	VAR robtarget Openhole_4834 := [[446.33, -4.29, 181.85], [-0.058838, 0.704655, 0.706057, -0.038517], [0,0,0,0], [9E9, 9E9, 9E9, 9E9, 9E9, 9E9]];
	VAR robtarget Openhole_4835 := [[445.84, -4.38, 181.92], [-0.060204, 0.704539, 0.70616, -0.036572], [0,0,0,0], [9E9, 9E9, 9E9, 9E9, 9E9, 9E9]];
	VAR robtarget Openhole_4836 := [[444.87, -4.57, 182.04], [-0.062827, 0.70431, 0.706355, -0.032605], [0,0,0,0], [9E9, 9E9, 9E9, 9E9, 9E9, 9E9]];
	VAR robtarget Openhole_4837 := [[438.56, -5.94, 182.78], [-0.079375, 0.702638, 0.707077, -0.006541], [0,0,0,0], [9E9, 9E9, 9E9, 9E9, 9E9, 9E9]];
	VAR robtarget Openhole_4838 := [[432.17, -6.93, 183.42], [-0.097021, 0.700419, 0.706868, 0.018385], [0,0,0,0], [9E9, 9E9, 9E9, 9E9, 9E9, 9E9]];
	VAR robtarget Openhole_4839 := [[431.68, -6.99, 183.47], [-0.09841, 0.700225, 0.706817, 0.020252], [0,0,0,0], [9E9, 9E9, 9E9, 9E9, 9E9, 9E9]];
	VAR robtarget Openhole_4840 := [[437.22, -4.54, 183.11], [-0.088439, 0.701554, 0.707076, -0.00665], [0,0,0,0], [9E9, 9E9, 9E9, 9E9, 9E9, 9E9]];
	VAR robtarget Openhole_4841 := [[442.51, -3.16, 182.47], [-0.075483, 0.703066, 0.706502, -0.029244], [0,0,0,0], [9E9, 9E9, 9E9, 9E9, 9E9, 9E9]];
	VAR robtarget Openhole_4842 := [[444.89, -2.47, 182.13], [-0.069759, 0.703657, 0.705995, -0.039633], [0,0,0,0], [9E9, 9E9, 9E9, 9E9, 9E9, 9E9]];
	VAR robtarget Openhole_4843 := [[445.84, -2.22, 181.99], [-0.067345, 0.703893, 0.705754, -0.043713], [0,0,0,0], [9E9, 9E9, 9E9, 9E9, 9E9, 9E9]];
	VAR robtarget Openhole_4844 := [[446.81, -2.01, 181.84], [-0.064778, 0.704133, 0.705496, -0.047696], [0,0,0,0], [9E9, 9E9, 9E9, 9E9, 9E9, 9E9]];
	VAR robtarget Openhole_4845 := [[447.3, -1.93, 181.76], [-0.063421, 0.704257, 0.705363, -0.049635], [0,0,0,0], [9E9, 9E9, 9E9, 9E9, 9E9, 9E9]];
	VAR robtarget Openhole_4846 := [[447.78, -1.85, 181.68], [-0.06202, 0.704382, 0.705226, -0.051544], [0,0,0,0], [9E9, 9E9, 9E9, 9E9, 9E9, 9E9]];
	VAR robtarget Openhole_4847 := [[448.27, -1.79, 181.6], [-0.060567, 0.704508, 0.705087, -0.053411], [0,0,0,0], [9E9, 9E9, 9E9, 9E9, 9E9, 9E9]];
	VAR robtarget Openhole_4848 := [[448.77, -1.75, 181.52], [-0.059016, 0.70464, 0.704949, -0.055201], [0,0,0,0], [9E9, 9E9, 9E9, 9E9, 9E9, 9E9]];
	VAR robtarget Openhole_4849 := [[449.26, -1.74, 181.44], [-0.057379, 0.704775, 0.704813, -0.056912], [0,0,0,0], [9E9, 9E9, 9E9, 9E9, 9E9, 9E9]];
	VAR robtarget Openhole_4850 := [[449.75, -1.74, 181.35], [-0.055693, 0.70491, 0.704677, -0.058572], [0,0,0,0], [9E9, 9E9, 9E9, 9E9, 9E9, 9E9]];
	VAR robtarget Openhole_4851 := [[450.24, -1.78, 181.27], [-0.053891, 0.70505, 0.704547, -0.060109], [0,0,0,0], [9E9, 9E9, 9E9, 9E9, 9E9, 9E9]];
	VAR robtarget Openhole_4852 := [[450.74, -1.83, 181.19], [-0.05205, 0.705189, 0.704419, -0.061598], [0,0,0,0], [9E9, 9E9, 9E9, 9E9, 9E9, 9E9]];
	VAR robtarget Openhole_4853 := [[451.22, -1.9, 181.11], [-0.050156, 0.705326, 0.704293, -0.063023], [0,0,0,0], [9E9, 9E9, 9E9, 9E9, 9E9, 9E9]];
	VAR robtarget Openhole_4854 := [[456.58, -2.86, 180.3], [-0.028679, 0.706525, 0.702811, -0.077823], [0,0,0,0], [9E9, 9E9, 9E9, 9E9, 9E9, 9E9]];
	VAR robtarget Openhole_4855 := [[458.54, -3.07, 180.01], [-0.021229, 0.706788, 0.702142, -0.083644], [0,0,0,0], [9E9, 9E9, 9E9, 9E9, 9E9, 9E9]];
	VAR robtarget Openhole_4856 := [[459.53, -3.13, 179.86], [-0.01766, 0.706886, 0.701769, -0.086718], [0,0,0,0], [9E9, 9E9, 9E9, 9E9, 9E9, 9E9]];
	VAR robtarget Openhole_4857 := [[460.52, -3.16, 179.71], [-0.014191, 0.706964, 0.701371, -0.089885], [0,0,0,0], [9E9, 9E9, 9E9, 9E9, 9E9, 9E9]];
	VAR robtarget Openhole_4858 := [[461.02, -3.16, 179.64], [-0.012499, 0.706996, 0.701161, -0.091504], [0,0,0,0], [9E9, 9E9, 9E9, 9E9, 9E9, 9E9]];
	VAR robtarget Openhole_4859 := [[461.51, -3.15, 179.56], [-0.010815, 0.707024, 0.700947, -0.093127], [0,0,0,0], [9E9, 9E9, 9E9, 9E9, 9E9, 9E9]];
	VAR robtarget Openhole_4860 := [[466.44, -2.87, 178.76], [0.005029, 0.707089, 0.6985, -0.109988], [0,0,0,0], [9E9, 9E9, 9E9, 9E9, 9E9, 9E9]];
	VAR robtarget Openhole_4861 := [[473.81, -2.37, 177.5], [0.028255, 0.706542, 0.69417, -0.13464], [0,0,0,0], [9E9, 9E9, 9E9, 9E9, 9E9, 9E9]];
	VAR robtarget Openhole_4862 := [[476.77, -2.31, 177.01], [0.037899, 0.70609, 0.692338, -0.143766], [0,0,0,0], [9E9, 9E9, 9E9, 9E9, 9E9, 9E9]];
	VAR robtarget Openhole_4863 := [[477.26, -2.32, 176.93], [0.039535, 0.706001, 0.692031, -0.145236], [0,0,0,0], [9E9, 9E9, 9E9, 9E9, 9E9, 9E9]];
	VAR robtarget Openhole_4864 := [[482.7, -2.51, 176.12], [0.05787, 0.704735, 0.688645, -0.160526], [0,0,0,0], [9E9, 9E9, 9E9, 9E9, 9E9, 9E9]];
	VAR robtarget Openhole_4865 := [[489.12, -3.09, 175.32], [0.079987, 0.702568, 0.684666, -0.176726], [0,0,0,0], [9E9, 9E9, 9E9, 9E9, 9E9, 9E9]];
	VAR robtarget Openhole_4866 := [[495.54, -3.95, 174.71], [0.102089, 0.699698, 0.680767, -0.191199], [0,0,0,0], [9E9, 9E9, 9E9, 9E9, 9E9, 9E9]];
	VAR robtarget Openhole_4867 := [[495.59, -2.66, 174.13], [0.098369, 0.700231, 0.679658, -0.195101], [0,0,0,0], [9E9, 9E9, 9E9, 9E9, 9E9, 9E9]];
	VAR robtarget Openhole_4868 := [[489.19, -1.71, 174.77], [0.075928, 0.703018, 0.683527, -0.181082], [0,0,0,0], [9E9, 9E9, 9E9, 9E9, 9E9, 9E9]];
	VAR robtarget Openhole_4869 := [[483.28, -1.11, 175.57], [0.055318, 0.70494, 0.68723, -0.166476], [0,0,0,0], [9E9, 9E9, 9E9, 9E9, 9E9, 9E9]];
	VAR robtarget Openhole_4870 := [[477.85, -0.87, 176.44], [0.036842, 0.706146, 0.690683, -0.151515], [0,0,0,0], [9E9, 9E9, 9E9, 9E9, 9E9, 9E9]];
	VAR robtarget Openhole_4871 := [[476.87, -0.86, 176.61], [0.033562, 0.70631, 0.691313, -0.148613], [0,0,0,0], [9E9, 9E9, 9E9, 9E9, 9E9, 9E9]];
	VAR robtarget Openhole_4872 := [[476.37, -0.86, 176.69], [0.031934, 0.706385, 0.691629, -0.147139], [0,0,0,0], [9E9, 9E9, 9E9, 9E9, 9E9, 9E9]];
	VAR robtarget Openhole_4873 := [[470.48, -1.08, 177.77], [0.012862, 0.70699, 0.695336, -0.128482], [0,0,0,0], [9E9, 9E9, 9E9, 9E9, 9E9, 9E9]];
	VAR robtarget Openhole_4874 := [[462.62, -1.59, 179.19], [-0.012185, 0.707002, 0.699732, -0.10186], [0,0,0,0], [9E9, 9E9, 9E9, 9E9, 9E9, 9E9]];
	VAR robtarget Openhole_4875 := [[461.64, -1.61, 179.36], [-0.015476, 0.706937, 0.700202, -0.098575], [0,0,0,0], [9E9, 9E9, 9E9, 9E9, 9E9, 9E9]];
	VAR robtarget Openhole_4876 := [[461.14, -1.61, 179.44], [-0.017156, 0.706899, 0.700428, -0.096959], [0,0,0,0], [9E9, 9E9, 9E9, 9E9, 9E9, 9E9]];
	VAR robtarget Openhole_4877 := [[460.65, -1.61, 179.53], [-0.018855, 0.706855, 0.700648, -0.095356], [0,0,0,0], [9E9, 9E9, 9E9, 9E9, 9E9, 9E9]];
	VAR robtarget Openhole_4878 := [[460.16, -1.6, 179.61], [-0.020577, 0.706807, 0.700861, -0.093773], [0,0,0,0], [9E9, 9E9, 9E9, 9E9, 9E9, 9E9]];
	VAR robtarget Openhole_4879 := [[459.17, -1.56, 179.77], [-0.024104, 0.706696, 0.701268, -0.09068], [0,0,0,0], [9E9, 9E9, 9E9, 9E9, 9E9, 9E9]];
	VAR robtarget Openhole_4880 := [[457.2, -1.38, 180.09], [-0.031441, 0.706407, 0.702007, -0.084775], [0,0,0,0], [9E9, 9E9, 9E9, 9E9, 9E9, 9E9]];
	VAR robtarget Openhole_4881 := [[454.77, -0.99, 180.48], [-0.04106, 0.705914, 0.702801, -0.077911], [0,0,0,0], [9E9, 9E9, 9E9, 9E9, 9E9, 9E9]];
	VAR robtarget Openhole_4882 := [[453.8, -0.8, 180.64], [-0.045008, 0.705673, 0.703086, -0.075301], [0,0,0,0], [9E9, 9E9, 9E9, 9E9, 9E9, 9E9]];
	VAR robtarget Openhole_4883 := [[452.84, -0.58, 180.8], [-0.049026, 0.705405, 0.703349, -0.0728], [0,0,0,0], [9E9, 9E9, 9E9, 9E9, 9E9, 9E9]];
	VAR robtarget Openhole_4884 := [[451.9, -0.27, 180.96], [-0.053242, 0.705099, 0.703568, -0.070651], [0,0,0,0], [9E9, 9E9, 9E9, 9E9, 9E9, 9E9]];
	VAR robtarget Openhole_4885 := [[451.43, -0.1, 181.04], [-0.055377, 0.704935, 0.703669, -0.069639], [0,0,0,0], [9E9, 9E9, 9E9, 9E9, 9E9, 9E9]];
	VAR robtarget Openhole_4886 := [[450.48, 0.12, 181.21], [-0.059395, 0.704608, 0.703911, -0.067156], [0,0,0,0], [9E9, 9E9, 9E9, 9E9, 9E9, 9E9]];
	VAR robtarget Openhole_4887 := [[449.49, 0.16, 181.39], [-0.062852, 0.704308, 0.704209, -0.063946], [0,0,0,0], [9E9, 9E9, 9E9, 9E9, 9E9, 9E9]];
	VAR robtarget Openhole_4888 := [[448.52, 0, 181.57], [-0.065623, 0.704055, 0.704545, -0.060131], [0,0,0,0], [9E9, 9E9, 9E9, 9E9, 9E9, 9E9]];
	VAR robtarget Openhole_4889 := [[448.05, -0.13, 181.66], [-0.066822, 0.703942, 0.704716, -0.058103], [0,0,0,0], [9E9, 9E9, 9E9, 9E9, 9E9, 9E9]];
	VAR robtarget Openhole_4890 := [[447.57, -0.24, 181.74], [-0.068056, 0.703824, 0.704878, -0.056092], [0,0,0,0], [9E9, 9E9, 9E9, 9E9, 9E9, 9E9]];
	VAR robtarget Openhole_4891 := [[447.09, -0.38, 181.83], [-0.069208, 0.703712, 0.705039, -0.054033], [0,0,0,0], [9E9, 9E9, 9E9, 9E9, 9E9, 9E9]];
	VAR robtarget Openhole_4892 := [[446.14, -0.63, 181.99], [-0.071596, 0.703473, 0.70534, -0.049958], [0,0,0,0], [9E9, 9E9, 9E9, 9E9, 9E9, 9E9]];
	VAR robtarget Openhole_4893 := [[445.19, -0.91, 182.15], [-0.073903, 0.703234, 0.70562, -0.045831], [0,0,0,0], [9E9, 9E9, 9E9, 9E9, 9E9, 9E9]];
	VAR robtarget Openhole_4894 := [[439.03, -2.77, 183.04], [-0.088301, 0.701572, 0.706861, -0.01864], [0,0,0,0], [9E9, 9E9, 9E9, 9E9, 9E9, 9E9]];
	VAR robtarget Openhole_4895 := [[441.88, -4.7, 182.45], [-0.072446, 0.703386, 0.706765, -0.021976], [0,0,0,0], [9E9, 9E9, 9E9, 9E9, 9E9, 9E9]];
	VAR robtarget Openhole_4896 := [[444.74, -6.64, 181.97], [-0.056353, 0.704858, 0.706655, -0.025274], [0,0,0,0], [9E9, 9E9, 9E9, 9E9, 9E9, 9E9]];
	VAR robtarget Openhole_4897 := [[445.24, -6.56, 181.91], [-0.054946, 0.704969, 0.706583, -0.027199], [0,0,0,0], [9E9, 9E9, 9E9, 9E9, 9E9, 9E9]];
	VAR robtarget Openhole_4898 := [[446.22, -6.44, 181.8], [-0.052032, 0.70519, 0.706428, -0.030973], [0,0,0,0], [9E9, 9E9, 9E9, 9E9, 9E9, 9E9]];
	VAR robtarget Openhole_4899 := [[447.21, -6.37, 181.68], [-0.048911, 0.705413, 0.706261, -0.034578], [0,0,0,0], [9E9, 9E9, 9E9, 9E9, 9E9, 9E9]];
	VAR robtarget Openhole_4900 := [[447.71, -6.35, 181.62], [-0.047279, 0.705524, 0.706174, -0.036316], [0,0,0,0], [9E9, 9E9, 9E9, 9E9, 9E9, 9E9]];
	VAR robtarget Openhole_4901 := [[448.2, -6.35, 181.56], [-0.045615, 0.705634, 0.706084, -0.038024], [0,0,0,0], [9E9, 9E9, 9E9, 9E9, 9E9, 9E9]];
	VAR robtarget Openhole_4902 := [[449.69, -6.4, 181.38], [-0.040367, 0.705954, 0.705805, -0.042891], [0,0,0,0], [9E9, 9E9, 9E9, 9E9, 9E9, 9E9]];
	VAR robtarget Openhole_4903 := [[452.66, -6.67, 181.03], [-0.029349, 0.706497, 0.70519, -0.052034], [0,0,0,0], [9E9, 9E9, 9E9, 9E9, 9E9, 9E9]];
	VAR robtarget Openhole_4904 := [[453.65, -6.78, 180.91], [-0.02559, 0.706644, 0.704966, -0.054976], [0,0,0,0], [9E9, 9E9, 9E9, 9E9, 9E9, 9E9]];
	VAR robtarget Openhole_4905 := [[454.64, -6.86, 180.8], [-0.021943, 0.706766, 0.70472, -0.058046], [0,0,0,0], [9E9, 9E9, 9E9, 9E9, 9E9, 9E9]];
	VAR robtarget Openhole_4906 := [[457.01, -8.37, 180.64], [-0.008792, 0.707052, 0.704474, -0.060967], [0,0,0,0], [9E9, 9E9, 9E9, 9E9, 9E9, 9E9]];
	VAR robtarget Openhole_4907 := [[455.02, -8.48, 180.85], [-0.015198, 0.706943, 0.705047, -0.053936], [0,0,0,0], [9E9, 9E9, 9E9, 9E9, 9E9, 9E9]];
	VAR robtarget Openhole_4908 := [[454.03, -8.5, 180.95], [-0.018531, 0.706864, 0.705299, -0.050525], [0,0,0,0], [9E9, 9E9, 9E9, 9E9, 9E9, 9E9]];
	VAR robtarget Openhole_4909 := [[453.53, -8.5, 181], [-0.020235, 0.706817, 0.705417, -0.048853], [0,0,0,0], [9E9, 9E9, 9E9, 9E9, 9E9, 9E9]];
	VAR robtarget Openhole_4910 := [[453.03, -8.5, 181.05], [-0.021918, 0.706767, 0.705532, -0.04716], [0,0,0,0], [9E9, 9E9, 9E9, 9E9, 9E9, 9E9]];
	VAR robtarget Openhole_4911 := [[452.53, -8.5, 181.1], [-0.023611, 0.706712, 0.705643, -0.045473], [0,0,0,0], [9E9, 9E9, 9E9, 9E9, 9E9, 9E9]];
	VAR robtarget Openhole_4912 := [[452.04, -8.5, 181.15], [-0.025316, 0.706653, 0.705749, -0.043799], [0,0,0,0], [9E9, 9E9, 9E9, 9E9, 9E9, 9E9]];
	VAR robtarget Openhole_4913 := [[447.06, -8.37, 181.66], [-0.042692, 0.705817, 0.706577, -0.027369], [0,0,0,0], [9E9, 9E9, 9E9, 9E9, 9E9, 9E9]];
	VAR robtarget Openhole_4914 := [[446.57, -8.37, 181.71], [-0.04439, 0.705712, 0.70664, -0.025688], [0,0,0,0], [9E9, 9E9, 9E9, 9E9, 9E9, 9E9]];
	VAR robtarget Openhole_4915 := [[446.07, -8.37, 181.76], [-0.046062, 0.705605, 0.7067, -0.023981], [0,0,0,0], [9E9, 9E9, 9E9, 9E9, 9E9, 9E9]];
	VAR robtarget Openhole_4916 := [[445.07, -8.4, 181.86], [-0.049339, 0.705383, 0.706809, -0.020506], [0,0,0,0], [9E9, 9E9, 9E9, 9E9, 9E9, 9E9]];
	VAR robtarget Openhole_4917 := [[444.58, -8.42, 181.91], [-0.050931, 0.70527, 0.706859, -0.018726], [0,0,0,0], [9E9, 9E9, 9E9, 9E9, 9E9, 9E9]];
	VAR robtarget Openhole_4918 := [[438.63, -8.96, 182.46], [-0.069107, 0.703722, 0.707099, 0.003299], [0,0,0,0], [9E9, 9E9, 9E9, 9E9, 9E9, 9E9]];
	VAR robtarget Openhole_4919 := [[437.22, -10.53, 182.41], [-0.068537, 0.703777, 0.706981, 0.013331], [0,0,0,0], [9E9, 9E9, 9E9, 9E9, 9E9, 9E9]];
	VAR robtarget Openhole_4920 := [[437.72, -10.53, 182.37], [-0.066866, 0.703938, 0.707011, 0.011663], [0,0,0,0], [9E9, 9E9, 9E9, 9E9, 9E9, 9E9]];
	VAR robtarget Openhole_4921 := [[438.21, -10.53, 182.33], [-0.065207, 0.704094, 0.707036, 0.009976], [0,0,0,0], [9E9, 9E9, 9E9, 9E9, 9E9, 9E9]];
	VAR robtarget Openhole_4922 := [[438.71, -10.53, 182.29], [-0.063541, 0.704246, 0.707058, 0.008294], [0,0,0,0], [9E9, 9E9, 9E9, 9E9, 9E9, 9E9]];
	VAR robtarget Openhole_4923 := [[439.21, -10.53, 182.25], [-0.061876, 0.704394, 0.707076, 0.006607], [0,0,0,0], [9E9, 9E9, 9E9, 9E9, 9E9, 9E9]];
	VAR robtarget Openhole_4924 := [[439.71, -10.53, 182.21], [-0.060221, 0.704538, 0.70709, 0.004907], [0,0,0,0], [9E9, 9E9, 9E9, 9E9, 9E9, 9E9]];
	VAR robtarget Openhole_4925 := [[442.7, -10.49, 181.97], [-0.050308, 0.705315, 0.707086, -0.005379], [0,0,0,0], [9E9, 9E9, 9E9, 9E9, 9E9, 9E9]];
	VAR robtarget Openhole_4926 := [[443.7, -10.51, 181.88], [-0.046878, 0.705551, 0.707053, -0.0087], [0,0,0,0], [9E9, 9E9, 9E9, 9E9, 9E9, 9E9]];
	VAR robtarget Openhole_4927 := [[444.19, -10.54, 181.84], [-0.045098, 0.705667, 0.707032, -0.010293], [0,0,0,0], [9E9, 9E9, 9E9, 9E9, 9E9, 9E9]];
	VAR robtarget Openhole_4928 := [[444.69, -10.59, 181.8], [-0.043247, 0.705783, 0.707008, -0.011805], [0,0,0,0], [9E9, 9E9, 9E9, 9E9, 9E9, 9E9]];
	VAR robtarget Openhole_4929 := [[445.18, -10.67, 181.76], [-0.041308, 0.705899, 0.706984, -0.013202], [0,0,0,0], [9E9, 9E9, 9E9, 9E9, 9E9, 9E9]];
	VAR robtarget Openhole_4930 := [[446.16, -10.86, 181.67], [-0.037367, 0.706119, 0.706928, -0.015916], [0,0,0,0], [9E9, 9E9, 9E9, 9E9, 9E9, 9E9]];
	VAR robtarget Openhole_4931 := [[446.72, -11.14, 181.62], [-0.03449, 0.706265, 0.706906, -0.016844], [0,0,0,0], [9E9, 9E9, 9E9, 9E9, 9E9, 9E9]];
	VAR robtarget Openhole_4932 := [[453.3, -11.75, 181.14], [-0.009998, 0.707036, 0.70613, -0.037151], [0,0,0,0], [9E9, 9E9, 9E9, 9E9, 9E9, 9E9]];
	VAR robtarget Openhole_4933 := [[453.93, -11.26, 181.08], [-0.009499, 0.707043, 0.705923, -0.0409], [0,0,0,0], [9E9, 9E9, 9E9, 9E9, 9E9, 9E9]];
	VAR robtarget Openhole_4934 := [[454.39, -11.08, 181.04], [-0.008559, 0.707055, 0.705793, -0.043089], [0,0,0,0], [9E9, 9E9, 9E9, 9E9, 9E9, 9E9]];
	VAR robtarget Openhole_4935 := [[454.86, -10.92, 180.99], [-0.007493, 0.707067, 0.705659, -0.045218], [0,0,0,0], [9E9, 9E9, 9E9, 9E9, 9E9, 9E9]];
	VAR robtarget Openhole_4936 := [[455.82, -10.65, 180.9], [-0.005139, 0.707088, 0.705382, -0.049354], [0,0,0,0], [9E9, 9E9, 9E9, 9E9, 9E9, 9E9]];
	VAR robtarget Openhole_4937 := [[456.31, -10.53, 180.85], [-0.003893, 0.707096, 0.705238, -0.051379], [0,0,0,0], [9E9, 9E9, 9E9, 9E9, 9E9, 9E9]];
	VAR robtarget Openhole_4938 := [[456.79, -10.4, 180.8], [-0.002687, 0.707102, 0.705086, -0.053422], [0,0,0,0], [9E9, 9E9, 9E9, 9E9, 9E9, 9E9]];
	VAR robtarget Openhole_4939 := [[457.75, -10.16, 180.7], [-0.000181, 0.707107, 0.704769, -0.057448], [0,0,0,0], [9E9, 9E9, 9E9, 9E9, 9E9, 9E9]];
	VAR robtarget Openhole_4940 := [[466.46, -8.15, 179.63], [0.022595, 0.706746, 0.700992, -0.092794], [0,0,0,0], [9E9, 9E9, 9E9, 9E9, 9E9, 9E9]];
	VAR robtarget Openhole_4941 := [[468.4, -7.76, 179.35], [0.027829, 0.706559, 0.699955, -0.100315], [0,0,0,0], [9E9, 9E9, 9E9, 9E9, 9E9, 9E9]];
	VAR robtarget Openhole_4942 := [[465.51, -9.96, 180.01], [0.025418, 0.70665, 0.702132, -0.08373], [0,0,0,0], [9E9, 9E9, 9E9, 9E9, 9E9, 9E9]];
	VAR robtarget Openhole_4943 := [[464.08, -10.39, 180.2], [0.022052, 0.706763, 0.70283, -0.077651], [0,0,0,0], [9E9, 9E9, 9E9, 9E9, 9E9, 9E9]];
	VAR robtarget Openhole_4944 := [[461.73, -11.18, 180.49], [0.016727, 0.706909, 0.703899, -0.067274], [0,0,0,0], [9E9, 9E9, 9E9, 9E9, 9E9, 9E9]];
	VAR robtarget Openhole_4945 := [[459.4, -12.06, 180.75], [0.011838, 0.707008, 0.704839, -0.056584], [0,0,0,0], [9E9, 9E9, 9E9, 9E9, 9E9, 9E9]];
	VAR robtarget Openhole_4946 := [[458.49, -12.46, 180.84], [0.010085, 0.707035, 0.705178, -0.052197], [0,0,0,0], [9E9, 9E9, 9E9, 9E9, 9E9, 9E9]];
	VAR robtarget Openhole_4947 := [[457.59, -12.89, 180.93], [0.008494, 0.707056, 0.705494, -0.047737], [0,0,0,0], [9E9, 9E9, 9E9, 9E9, 9E9, 9E9]];
	VAR robtarget Openhole_4948 := [[457.15, -13.13, 180.98], [0.007804, 0.707064, 0.705643, -0.045469], [0,0,0,0], [9E9, 9E9, 9E9, 9E9, 9E9, 9E9]];
	VAR robtarget Openhole_4949 := [[456.74, -13.4, 181.02], [0.007289, 0.707069, 0.705789, -0.043151], [0,0,0,0], [9E9, 9E9, 9E9, 9E9, 9E9, 9E9]];
	VAR robtarget Openhole_4950 := [[456.33, -13.69, 181.06], [0.006906, 0.707073, 0.705928, -0.040806], [0,0,0,0], [9E9, 9E9, 9E9, 9E9, 9E9, 9E9]];
	VAR robtarget Openhole_4951 := [[455.86, -14.06, 181.11], [0.006573, 0.707076, 0.706086, -0.037975], [0,0,0,0], [9E9, 9E9, 9E9, 9E9, 9E9, 9E9]];
	VAR robtarget Openhole_4952 := [[443.92, -12.82, 181.75], [-0.038296, 0.706069, 0.707105, -0.001664], [0,0,0,0], [9E9, 9E9, 9E9, 9E9, 9E9, 9E9]];
	VAR robtarget Openhole_4953 := [[443.19, -12.46, 181.81], [-0.041996, 0.705859, 0.707107, -0.000403], [0,0,0,0], [9E9, 9E9, 9E9, 9E9, 9E9, 9E9]];
	VAR robtarget Openhole_4954 := [[442.2, -12.35, 181.88], [-0.045717, 0.705627, 0.707102, 0.002592], [0,0,0,0], [9E9, 9E9, 9E9, 9E9, 9E9, 9E9]];
	VAR robtarget Openhole_4955 := [[441.7, -12.31, 181.92], [-0.047524, 0.705508, 0.707095, 0.004149], [0,0,0,0], [9E9, 9E9, 9E9, 9E9, 9E9, 9E9]];
	VAR robtarget Openhole_4956 := [[440.21, -12.22, 182.02], [-0.052839, 0.70513, 0.70705, 0.008925], [0,0,0,0], [9E9, 9E9, 9E9, 9E9, 9E9, 9E9]];
	VAR robtarget Openhole_4957 := [[439.21, -12.15, 182.09], [-0.056421, 0.704852, 0.707004, 0.012046], [0,0,0,0], [9E9, 9E9, 9E9, 9E9, 9E9, 9E9]];
	VAR robtarget Openhole_4958 := [[438.22, -12.1, 182.16], [-0.059936, 0.704562, 0.706943, 0.015229], [0,0,0,0], [9E9, 9E9, 9E9, 9E9, 9E9, 9E9]];
	VAR robtarget Openhole_4959 := [[435.3, -16.15, 181.81], [-0.055995, 0.704886, 0.706049, 0.038666], [0,0,0,0], [9E9, 9E9, 9E9, 9E9, 9E9, 9E9]];
	VAR robtarget Openhole_4960 := [[434.81, -16.09, 181.83], [-0.057843, 0.704737, 0.705967, 0.040124], [0,0,0,0], [9E9, 9E9, 9E9, 9E9, 9E9, 9E9]];
	VAR robtarget Openhole_4961 := [[433.81, -16, 181.87], [-0.061461, 0.704431, 0.705791, 0.043121], [0,0,0,0], [9E9, 9E9, 9E9, 9E9, 9E9, 9E9]];
	VAR robtarget Openhole_4962 := [[425.83, -15.62, 182.19], [-0.088741, 0.701516, 0.703821, 0.068084], [0,0,0,0], [9E9, 9E9, 9E9, 9E9, 9E9, 9E9]];
	VAR robtarget Openhole_4963 := [[411.84, -15.42, 182.72], [-0.132375, 0.694606, 0.69832, 0.111126], [0,0,0,0], [9E9, 9E9, 9E9, 9E9, 9E9, 9E9]];
	VAR robtarget Openhole_4964 := [[411.34, -15.42, 182.74], [-0.133839, 0.694325, 0.698081, 0.112621], [0,0,0,0], [9E9, 9E9, 9E9, 9E9, 9E9, 9E9]];
	VAR robtarget Openhole_4965 := [[410.84, -15.42, 182.76], [-0.135296, 0.694043, 0.697838, 0.114113], [0,0,0,0], [9E9, 9E9, 9E9, 9E9, 9E9, 9E9]];
	VAR robtarget Openhole_4966 := [[399.85, -15.62, 183.04], [-0.165401, 0.68749, 0.691832, 0.146179], [0,0,0,0], [9E9, 9E9, 9E9, 9E9, 9E9, 9E9]];
	VAR robtarget Openhole_4967 := [[394.35, -15.88, 183.09], [-0.178974, 0.684082, 0.688381, 0.161652], [0,0,0,0], [9E9, 9E9, 9E9, 9E9, 9E9, 9E9]];
	VAR robtarget Openhole_4968 := [[389.35, -15.88, 183.24], [-0.191413, 0.680706, 0.685251, 0.174443], [0,0,0,0], [9E9, 9E9, 9E9, 9E9, 9E9, 9E9]];
	VAR robtarget Openhole_4969 := [[362.35, -15.88, 183.33], [-0.183051, 0.683002, 0.683002, 0.183051], [0,0,0,0], [9E9, 9E9, 9E9, 9E9, 9E9, 9E9]];
	VAR robtarget Openhole_4970 := [[362.34, -21.09, 180.31], [-0.183051, 0.683002, 0.683002, 0.183051], [0,0,0,0], [9E9, 9E9, 9E9, 9E9, 9E9, 9E9]];
	VAR robtarget Openhole_4971 := [[389.34, -21.09, 180.23], [-0.176562, 0.684709, 0.681301, 0.189286], [0,0,0,0], [9E9, 9E9, 9E9, 9E9, 9E9, 9E9]];
	VAR robtarget Openhole_4972 := [[394.34, -21.09, 180.33], [-0.163743, 0.687887, 0.684629, 0.176869], [0,0,0,0], [9E9, 9E9, 9E9, 9E9, 9E9, 9E9]];
	VAR robtarget Openhole_4973 := [[395.21, -21.06, 180.36], [-0.161544, 0.688407, 0.685224, 0.174552], [0,0,0,0], [9E9, 9E9, 9E9, 9E9, 9E9, 9E9]];
	VAR robtarget Openhole_4974 := [[401.7, -20.78, 180.62], [-0.144771, 0.692128, 0.689543, 0.156624], [0,0,0,0], [9E9, 9E9, 9E9, 9E9, 9E9, 9E9]];
	VAR robtarget Openhole_4975 := [[406.7, -20.73, 180.72], [-0.130756, 0.694912, 0.692576, 0.142615], [0,0,0,0], [9E9, 9E9, 9E9, 9E9, 9E9, 9E9]];
	VAR robtarget Openhole_4976 := [[407.2, -20.73, 180.73], [-0.129307, 0.695183, 0.692865, 0.1412], [0,0,0,0], [9E9, 9E9, 9E9, 9E9, 9E9, 9E9]];
	VAR robtarget Openhole_4977 := [[421.2, -20.9, 180.91], [-0.086161, 0.701838, 0.699994, 0.10004], [0,0,0,0], [9E9, 9E9, 9E9, 9E9, 9E9, 9E9]];
	VAR robtarget Openhole_4978 := [[421.7, -20.9, 180.92], [-0.084573, 0.702031, 0.700215, 0.098481], [0,0,0,0], [9E9, 9E9, 9E9, 9E9, 9E9, 9E9]];
	VAR robtarget Openhole_4979 := [[425.2, -20.8, 181.01], [-0.073658, 0.70326, 0.701715, 0.087152], [0,0,0,0], [9E9, 9E9, 9E9, 9E9, 9E9, 9E9]];
	VAR robtarget Openhole_4980 := [[426.19, -20.74, 181.04], [-0.070639, 0.70357, 0.702129, 0.083758], [0,0,0,0], [9E9, 9E9, 9E9, 9E9, 9E9, 9E9]];
	VAR robtarget Openhole_4981 := [[428.18, -20.56, 181.11], [-0.064746, 0.704136, 0.702927, 0.076766], [0,0,0,0], [9E9, 9E9, 9E9, 9E9, 9E9, 9E9]];
	VAR robtarget Openhole_4982 := [[429.18, -20.43, 181.15], [-0.061923, 0.70439, 0.703315, 0.073135], [0,0,0,0], [9E9, 9E9, 9E9, 9E9, 9E9, 9E9]];
	VAR robtarget Openhole_4983 := [[429.67, -20.35, 181.17], [-0.060557, 0.704509, 0.703505, 0.071276], [0,0,0,0], [9E9, 9E9, 9E9, 9E9, 9E9, 9E9]];
	VAR robtarget Openhole_4984 := [[431.14, -20.07, 181.24], [-0.056638, 0.704835, 0.704063, 0.065543], [0,0,0,0], [9E9, 9E9, 9E9, 9E9, 9E9, 9E9]];
	VAR robtarget Openhole_4985 := [[433.09, -19.64, 181.33], [-0.051617, 0.70522, 0.704749, 0.057692], [0,0,0,0], [9E9, 9E9, 9E9, 9E9, 9E9, 9E9]];
	VAR robtarget Openhole_4986 := [[431.92, -18.36, 181.53], [-0.059796, 0.704574, 0.704786, 0.057245], [0,0,0,0], [9E9, 9E9, 9E9, 9E9, 9E9, 9E9]];
	VAR robtarget Openhole_4987 := [[431.43, -18.38, 181.53], [-0.061346, 0.704441, 0.704642, 0.058985], [0,0,0,0], [9E9, 9E9, 9E9, 9E9, 9E9, 9E9]];
	VAR robtarget Openhole_4988 := [[430.43, -18.38, 181.54], [-0.064643, 0.704146, 0.70436, 0.062263], [0,0,0,0], [9E9, 9E9, 9E9, 9E9, 9E9, 9E9]];
	VAR robtarget Openhole_4989 := [[426.43, -18.45, 181.55], [-0.077476, 0.70285, 0.703069, 0.075459], [0,0,0,0], [9E9, 9E9, 9E9, 9E9, 9E9, 9E9]];
	VAR robtarget Openhole_4990 := [[425.93, -18.44, 181.55], [-0.0791, 0.702669, 0.702895, 0.077058], [0,0,0,0], [9E9, 9E9, 9E9, 9E9, 9E9, 9E9]];
	VAR robtarget Openhole_4991 := [[408.43, -18.16, 181.76], [-0.133739, 0.694344, 0.695105, 0.129729], [0,0,0,0], [9E9, 9E9, 9E9, 9E9, 9E9, 9E9]];
	VAR robtarget Openhole_4992 := [[407.93, -18.16, 181.77], [-0.135183, 0.694065, 0.694833, 0.131174], [0,0,0,0], [9E9, 9E9, 9E9, 9E9, 9E9, 9E9]];
	VAR robtarget Openhole_4993 := [[398.93, -18.33, 181.76], [-0.159738, 0.688828, 0.689513, 0.156755], [0,0,0,0], [9E9, 9E9, 9E9, 9E9, 9E9, 9E9]];
	VAR robtarget Openhole_4994 := [[394.35, -18.56, 181.67], [-0.17115, 0.686081, 0.686493, 0.16949], [0,0,0,0], [9E9, 9E9, 9E9, 9E9, 9E9, 9E9]];
	VAR robtarget Openhole_4995 := [[362.35, -18.56, 181.78], [-0.183051, 0.683002, 0.683002, 0.183051], [0,0,0,0], [9E9, 9E9, 9E9, 9E9, 9E9, 9E9]];
	VAR robtarget Openhole_4996 := [[362.35, -17.6, 182.33], [-0.183051, 0.683002, 0.683002, 0.183051], [0,0,0,0], [9E9, 9E9, 9E9, 9E9, 9E9, 9E9]];
	VAR robtarget Openhole_4997 := [[389.35, -17.6, 182.25], [-0.186521, 0.682063, 0.683983, 0.179351], [0,0,0,0], [9E9, 9E9, 9E9, 9E9, 9E9, 9E9]];
	VAR robtarget Openhole_4998 := [[394.35, -17.6, 182.18], [-0.173956, 0.685375, 0.68718, 0.166684], [0,0,0,0], [9E9, 9E9, 9E9, 9E9, 9E9, 9E9]];
	VAR robtarget Openhole_4999 := [[403.05, -17.26, 182.21], [-0.15174, 0.690634, 0.692644, 0.142285], [0,0,0,0], [9E9, 9E9, 9E9, 9E9, 9E9, 9E9]];
	VAR robtarget Openhole_5000 := [[408.55, -17.2, 182.14], [-0.136393, 0.693828, 0.695715, 0.126416], [0,0,0,0], [9E9, 9E9, 9E9, 9E9, 9E9, 9E9]];
	VAR robtarget Openhole_5001 := [[409.05, -17.2, 182.13], [-0.134946, 0.694111, 0.695978, 0.12496], [0,0,0,0], [9E9, 9E9, 9E9, 9E9, 9E9, 9E9]];
	VAR robtarget Openhole_5002 := [[423.54, -17.43, 181.82], [-0.090067, 0.701347, 0.702408, 0.081382], [0,0,0,0], [9E9, 9E9, 9E9, 9E9, 9E9, 9E9]];
	VAR robtarget Openhole_5003 := [[433.04, -17.58, 181.65], [-0.058704, 0.704666, 0.705266, 0.050995], [0,0,0,0], [9E9, 9E9, 9E9, 9E9, 9E9, 9E9]];
	VAR robtarget Openhole_5004 := [[433.54, -17.58, 181.64], [-0.057068, 0.7048, 0.705385, 0.049318], [0,0,0,0], [9E9, 9E9, 9E9, 9E9, 9E9, 9E9]];
	VAR robtarget Openhole_5005 := [[434.04, -17.59, 181.63], [-0.055381, 0.704935, 0.705497, 0.047686], [0,0,0,0], [9E9, 9E9, 9E9, 9E9, 9E9, 9E9]];
	VAR robtarget Openhole_5006 := [[434.54, -17.58, 181.63], [-0.05373, 0.705062, 0.705608, 0.046012], [0,0,0,0], [9E9, 9E9, 9E9, 9E9, 9E9, 9E9]];
	VAR robtarget Openhole_5007 := [[435.04, -17.58, 181.62], [-0.052062, 0.705188, 0.705715, 0.044351], [0,0,0,0], [9E9, 9E9, 9E9, 9E9, 9E9, 9E9]];
	VAR robtarget Openhole_5008 := [[435.54, -17.56, 181.62], [-0.050458, 0.705304, 0.705821, 0.042623], [0,0,0,0], [9E9, 9E9, 9E9, 9E9, 9E9, 9E9]];
	VAR robtarget Openhole_5009 := [[436.54, -17.57, 181.6], [-0.047087, 0.705537, 0.706013, 0.039312], [0,0,0,0], [9E9, 9E9, 9E9, 9E9, 9E9, 9E9]];
	VAR robtarget Openhole_5010 := [[437.08, -18.86, 181.44], [-0.040922, 0.705922, 0.70587, 0.041808], [0,0,0,0], [9E9, 9E9, 9E9, 9E9, 9E9, 9E9]];
	VAR robtarget Openhole_5011 := [[436.63, -19.07, 181.42], [-0.041713, 0.705875, 0.705734, 0.044035], [0,0,0,0], [9E9, 9E9, 9E9, 9E9, 9E9, 9E9]];
	VAR robtarget Openhole_5012 := [[435.69, -19.42, 181.37], [-0.043687, 0.705756, 0.705454, 0.048321], [0,0,0,0], [9E9, 9E9, 9E9, 9E9, 9E9, 9E9]];
	VAR robtarget Openhole_5013 := [[434.78, -19.82, 181.31], [-0.045388, 0.705649, 0.70514, 0.052706], [0,0,0,0], [9E9, 9E9, 9E9, 9E9, 9E9, 9E9]];
	VAR robtarget Openhole_5014 := [[434.32, -20.01, 181.28], [-0.046293, 0.70559, 0.704975, 0.05487], [0,0,0,0], [9E9, 9E9, 9E9, 9E9, 9E9, 9E9]];
	VAR robtarget Openhole_5015 := [[433.85, -20.18, 181.25], [-0.047271, 0.705525, 0.704806, 0.056998], [0,0,0,0], [9E9, 9E9, 9E9, 9E9, 9E9, 9E9]];
	VAR robtarget Openhole_5016 := [[432.43, -20.64, 181.16], [-0.050465, 0.705304, 0.704274, 0.063232], [0,0,0,0], [9E9, 9E9, 9E9, 9E9, 9E9, 9E9]];
	VAR robtarget Openhole_5017 := [[430.02, -21.29, 181], [-0.056289, 0.704863, 0.703302, 0.073252], [0,0,0,0], [9E9, 9E9, 9E9, 9E9, 9E9, 9E9]];
	VAR robtarget Openhole_5018 := [[429.04, -21.5, 180.94], [-0.058776, 0.70466, 0.702888, 0.07713], [0,0,0,0], [9E9, 9E9, 9E9, 9E9, 9E9, 9E9]];
	VAR robtarget Openhole_5019 := [[428.06, -21.68, 180.88], [-0.061404, 0.704436, 0.702465, 0.080891], [0,0,0,0], [9E9, 9E9, 9E9, 9E9, 9E9, 9E9]];
	VAR robtarget Openhole_5020 := [[424.09, -22.12, 180.67], [-0.072896, 0.703339, 0.700702, 0.094958], [0,0,0,0], [9E9, 9E9, 9E9, 9E9, 9E9, 9E9]];
	VAR robtarget Openhole_5021 := [[423.09, -22.18, 180.62], [-0.075904, 0.703021, 0.700241, 0.098296], [0,0,0,0], [9E9, 9E9, 9E9, 9E9, 9E9, 9E9]];
	VAR robtarget Openhole_5022 := [[418.1, -22.26, 180.45], [-0.091497, 0.701162, 0.697858, 0.113995], [0,0,0,0], [9E9, 9E9, 9E9, 9E9, 9E9, 9E9]];
	VAR robtarget Openhole_5023 := [[417.6, -22.26, 180.43], [-0.093063, 0.700956, 0.697608, 0.11551], [0,0,0,0], [9E9, 9E9, 9E9, 9E9, 9E9, 9E9]];
	VAR robtarget Openhole_5024 := [[405.6, -22.12, 180.12], [-0.129614, 0.695126, 0.69102, 0.149969], [0,0,0,0], [9E9, 9E9, 9E9, 9E9, 9E9, 9E9]];
	VAR robtarget Openhole_5025 := [[405.1, -22.12, 180.1], [-0.131052, 0.694856, 0.690718, 0.151358], [0,0,0,0], [9E9, 9E9, 9E9, 9E9, 9E9, 9E9]];
	VAR robtarget Openhole_5026 := [[397.61, -22.29, 179.8], [-0.15148, 0.690691, 0.685875, 0.171976], [0,0,0,0], [9E9, 9E9, 9E9, 9E9, 9E9, 9E9]];
	VAR robtarget Openhole_5027 := [[395.12, -22.43, 179.64], [-0.157747, 0.689286, 0.684129, 0.178793], [0,0,0,0], [9E9, 9E9, 9E9, 9E9, 9E9, 9E9]];
	VAR robtarget Openhole_5028 := [[394.34, -22.46, 179.6], [-0.159728, 0.68883, 0.683588, 0.180853], [0,0,0,0], [9E9, 9E9, 9E9, 9E9, 9E9, 9E9]];
	VAR robtarget Openhole_5029 := [[389.34, -22.46, 179.44], [-0.172647, 0.685706, 0.68021, 0.193171], [0,0,0,0], [9E9, 9E9, 9E9, 9E9, 9E9, 9E9]];
	VAR robtarget Openhole_5030 := [[362.34, -22.46, 179.52], [-0.183051, 0.683002, 0.683002, 0.183051], [0,0,0,0], [9E9, 9E9, 9E9, 9E9, 9E9, 9E9]];
	VAR robtarget Openhole_5031 := [[362.34, -23.36, 179], [-0.183051, 0.683002, 0.683002, 0.183051], [0,0,0,0], [9E9, 9E9, 9E9, 9E9, 9E9, 9E9]];
	VAR robtarget Openhole_5032 := [[389.34, -23.36, 178.92], [-0.170067, 0.686351, 0.679479, 0.195724], [0,0,0,0], [9E9, 9E9, 9E9, 9E9, 9E9, 9E9]];
	VAR robtarget Openhole_5033 := [[394.34, -23.36, 179.13], [-0.157083, 0.689438, 0.68289, 0.183471], [0,0,0,0], [9E9, 9E9, 9E9, 9E9, 9E9, 9E9]];
	VAR robtarget Openhole_5034 := [[395.23, -23.34, 179.18], [-0.154791, 0.689956, 0.683507, 0.181156], [0,0,0,0], [9E9, 9E9, 9E9, 9E9, 9E9, 9E9]];
	VAR robtarget Openhole_5035 := [[401.21, -23.09, 179.54], [-0.13915, 0.69328, 0.687618, 0.164868], [0,0,0,0], [9E9, 9E9, 9E9, 9E9, 9E9, 9E9]];
	VAR robtarget Openhole_5036 := [[404.71, -23.06, 179.69], [-0.129304, 0.695184, 0.689841, 0.155302], [0,0,0,0], [9E9, 9E9, 9E9, 9E9, 9E9, 9E9]];
	VAR robtarget Openhole_5037 := [[405.21, -23.06, 179.71], [-0.12786, 0.695451, 0.690149, 0.153928], [0,0,0,0], [9E9, 9E9, 9E9, 9E9, 9E9, 9E9]];
	VAR robtarget Openhole_5038 := [[417.2, -23.21, 180.13], [-0.091251, 0.701194, 0.696894, 0.119745], [0,0,0,0], [9E9, 9E9, 9E9, 9E9, 9E9, 9E9]];
	VAR robtarget Openhole_5039 := [[417.7, -23.21, 180.15], [-0.089689, 0.701396, 0.697152, 0.118233], [0,0,0,0], [9E9, 9E9, 9E9, 9E9, 9E9, 9E9]];
	VAR robtarget Openhole_5040 := [[418.2, -23.21, 180.17], [-0.088119, 0.701595, 0.697407, 0.11672], [0,0,0,0], [9E9, 9E9, 9E9, 9E9, 9E9, 9E9]];
	VAR robtarget Openhole_5041 := [[418.7, -23.21, 180.19], [-0.086557, 0.701789, 0.697661, 0.115191], [0,0,0,0], [9E9, 9E9, 9E9, 9E9, 9E9, 9E9]];
	VAR robtarget Openhole_5042 := [[423.19, -23.06, 180.41], [-0.07271, 0.703359, 0.699877, 0.100855], [0,0,0,0], [9E9, 9E9, 9E9, 9E9, 9E9, 9E9]];
	VAR robtarget Openhole_5043 := [[425.18, -22.88, 180.52], [-0.066851, 0.70394, 0.700828, 0.094025], [0,0,0,0], [9E9, 9E9, 9E9, 9E9, 9E9, 9E9]];
	VAR robtarget Openhole_5044 := [[428.14, -22.45, 180.72], [-0.058589, 0.704675, 0.702199, 0.083168], [0,0,0,0], [9E9, 9E9, 9E9, 9E9, 9E9, 9E9]];
	VAR robtarget Openhole_5045 := [[428.63, -22.36, 180.76], [-0.057297, 0.704782, 0.70242, 0.081278], [0,0,0,0], [9E9, 9E9, 9E9, 9E9, 9E9, 9E9]];
	VAR robtarget Openhole_5046 := [[430.48, -23.42, 180.62], [-0.047648, 0.7055, 0.702701, 0.078812], [0,0,0,0], [9E9, 9E9, 9E9, 9E9, 9E9, 9E9]];
	VAR robtarget Openhole_5047 := [[429.52, -23.69, 180.53], [-0.049911, 0.705343, 0.702241, 0.082811], [0,0,0,0], [9E9, 9E9, 9E9, 9E9, 9E9, 9E9]];
	VAR robtarget Openhole_5048 := [[428.07, -24.05, 180.39], [-0.053486, 0.705081, 0.701526, 0.088665], [0,0,0,0], [9E9, 9E9, 9E9, 9E9, 9E9, 9E9]];
	VAR robtarget Openhole_5049 := [[427.1, -24.27, 180.3], [-0.055977, 0.704888, 0.701034, 0.092472], [0,0,0,0], [9E9, 9E9, 9E9, 9E9, 9E9, 9E9]];
	VAR robtarget Openhole_5050 := [[426.61, -24.36, 180.25], [-0.057271, 0.704784, 0.700786, 0.094335], [0,0,0,0], [9E9, 9E9, 9E9, 9E9, 9E9, 9E9]];
	VAR robtarget Openhole_5051 := [[425.14, -24.59, 180.12], [-0.061335, 0.704442, 0.700034, 0.099761], [0,0,0,0], [9E9, 9E9, 9E9, 9E9, 9E9, 9E9]];
	VAR robtarget Openhole_5052 := [[424.15, -24.72, 180.04], [-0.064144, 0.704191, 0.699525, 0.103271], [0,0,0,0], [9E9, 9E9, 9E9, 9E9, 9E9, 9E9]];
	VAR robtarget Openhole_5053 := [[419.67, -25.03, 179.71], [-0.077536, 0.702843, 0.697175, 0.118096], [0,0,0,0], [9E9, 9E9, 9E9, 9E9, 9E9, 9E9]];
	VAR robtarget Openhole_5054 := [[416.18, -25.08, 179.49], [-0.088411, 0.701558, 0.695285, 0.128761], [0,0,0,0], [9E9, 9E9, 9E9, 9E9, 9E9, 9E9]];
	VAR robtarget Openhole_5055 := [[415.68, -25.08, 179.46], [-0.089979, 0.701359, 0.69501, 0.130235], [0,0,0,0], [9E9, 9E9, 9E9, 9E9, 9E9, 9E9]];
	VAR robtarget Openhole_5056 := [[402.2, -24.86, 178.77], [-0.130975, 0.694871, 0.686972, 0.167539], [0,0,0,0], [9E9, 9E9, 9E9, 9E9, 9E9, 9E9]];
	VAR robtarget Openhole_5057 := [[401.7, -24.86, 178.75], [-0.132392, 0.694602, 0.686646, 0.168871], [0,0,0,0], [9E9, 9E9, 9E9, 9E9, 9E9, 9E9]];
	VAR robtarget Openhole_5058 := [[395.72, -25.05, 178.32], [-0.148426, 0.691353, 0.682508, 0.184885], [0,0,0,0], [9E9, 9E9, 9E9, 9E9, 9E9, 9E9]];
	VAR robtarget Openhole_5059 := [[395.22, -25.08, 178.27], [-0.149676, 0.691084, 0.682144, 0.186223], [0,0,0,0], [9E9, 9E9, 9E9, 9E9, 9E9, 9E9]];
	VAR robtarget Openhole_5060 := [[394.34, -25.1, 178.21], [-0.15199, 0.690579, 0.681519, 0.188499], [0,0,0,0], [9E9, 9E9, 9E9, 9E9, 9E9, 9E9]];
	VAR robtarget Openhole_5061 := [[389.34, -25.1, 177.91], [-0.165099, 0.687563, 0.678048, 0.200626], [0,0,0,0], [9E9, 9E9, 9E9, 9E9, 9E9, 9E9]];
	VAR robtarget Openhole_5062 := [[362.34, -25.1, 178], [-0.183051, 0.683002, 0.683002, 0.183051], [0,0,0,0], [9E9, 9E9, 9E9, 9E9, 9E9, 9E9]];
	VAR robtarget Openhole_5063 := [[362.33, -25.89, 177.54], [-0.183051, 0.683002, 0.683002, 0.183051], [0,0,0,0], [9E9, 9E9, 9E9, 9E9, 9E9, 9E9]];
	VAR robtarget Openhole_5064 := [[389.33, -25.89, 177.46], [-0.16285, 0.688099, 0.677389, 0.20284], [0,0,0,0], [9E9, 9E9, 9E9, 9E9, 9E9, 9E9]];
	VAR robtarget Openhole_5065 := [[394.33, -25.89, 177.79], [-0.149685, 0.691082, 0.680887, 0.190769], [0,0,0,0], [9E9, 9E9, 9E9, 9E9, 9E9, 9E9]];
	VAR robtarget Openhole_5066 := [[395.1, -25.86, 177.85], [-0.147682, 0.691513, 0.681436, 0.188797], [0,0,0,0], [9E9, 9E9, 9E9, 9E9, 9E9, 9E9]];
	VAR robtarget Openhole_5067 := [[400.58, -25.68, 178.3], [-0.133074, 0.694472, 0.685296, 0.174269], [0,0,0,0], [9E9, 9E9, 9E9, 9E9, 9E9, 9E9]];
	VAR robtarget Openhole_5068 := [[401.58, -25.68, 178.36], [-0.130255, 0.695006, 0.685961, 0.171633], [0,0,0,0], [9E9, 9E9, 9E9, 9E9, 9E9, 9E9]];
	VAR robtarget Openhole_5069 := [[402.08, -25.68, 178.4], [-0.128829, 0.695272, 0.686289, 0.170314], [0,0,0,0], [9E9, 9E9, 9E9, 9E9, 9E9, 9E9]];
	VAR robtarget Openhole_5070 := [[416.05, -25.98, 179.19], [-0.085938, 0.701865, 0.694682, 0.131973], [0,0,0,0], [9E9, 9E9, 9E9, 9E9, 9E9, 9E9]];
	VAR robtarget Openhole_5071 := [[416.55, -25.98, 179.23], [-0.084371, 0.702055, 0.694962, 0.130492], [0,0,0,0], [9E9, 9E9, 9E9, 9E9, 9E9, 9E9]];
	VAR robtarget Openhole_5072 := [[421.53, -25.83, 179.6], [-0.068981, 0.703734, 0.697699, 0.114959], [0,0,0,0], [9E9, 9E9, 9E9, 9E9, 9E9, 9E9]];
	VAR robtarget Openhole_5073 := [[425, -25.46, 179.91], [-0.058911, 0.704648, 0.699561, 0.103026], [0,0,0,0], [9E9, 9E9, 9E9, 9E9, 9E9, 9E9]];
	VAR robtarget Openhole_5074 := [[426.96, -25.13, 180.11], [-0.053576, 0.705074, 0.700595, 0.095744], [0,0,0,0], [9E9, 9E9, 9E9, 9E9, 9E9, 9E9]];
	VAR robtarget Openhole_5075 := [[427.45, -25.03, 180.16], [-0.052321, 0.705168, 0.70085, 0.093854], [0,0,0,0], [9E9, 9E9, 9E9, 9E9, 9E9, 9E9]];
	VAR robtarget Openhole_5076 := [[430.33, -24.25, 180.47], [-0.04537, 0.70565, 0.70233, 0.082055], [0,0,0,0], [9E9, 9E9, 9E9, 9E9, 9E9, 9E9]];
	VAR robtarget Openhole_5077 := [[430.8, -24.09, 180.52], [-0.04432, 0.705716, 0.702565, 0.080011], [0,0,0,0], [9E9, 9E9, 9E9, 9E9, 9E9, 9E9]];
	VAR robtarget Openhole_5078 := [[431.73, -23.75, 180.62], [-0.042364, 0.705837, 0.703028, 0.075838], [0,0,0,0], [9E9, 9E9, 9E9, 9E9, 9E9, 9E9]];
	VAR robtarget Openhole_5079 := [[432.19, -23.56, 180.67], [-0.041445, 0.705891, 0.703254, 0.073718], [0,0,0,0], [9E9, 9E9, 9E9, 9E9, 9E9, 9E9]];
	VAR robtarget Openhole_5080 := [[432.65, -23.37, 180.72], [-0.040566, 0.705942, 0.703475, 0.071577], [0,0,0,0], [9E9, 9E9, 9E9, 9E9, 9E9, 9E9]];
	VAR robtarget Openhole_5081 := [[433.55, -22.94, 180.83], [-0.038974, 0.706032, 0.703905, 0.067216], [0,0,0,0], [9E9, 9E9, 9E9, 9E9, 9E9, 9E9]];
	VAR robtarget Openhole_5082 := [[434, -22.72, 180.88], [-0.038241, 0.706072, 0.704112, 0.065008], [0,0,0,0], [9E9, 9E9, 9E9, 9E9, 9E9, 9E9]];
	VAR robtarget Openhole_5083 := [[434.43, -22.48, 180.93], [-0.037569, 0.706108, 0.704315, 0.062776], [0,0,0,0], [9E9, 9E9, 9E9, 9E9, 9E9, 9E9]];
	VAR robtarget Openhole_5084 := [[435.29, -21.98, 181.02], [-0.03636, 0.706171, 0.704703, 0.05826], [0,0,0,0], [9E9, 9E9, 9E9, 9E9, 9E9, 9E9]];
	VAR robtarget Openhole_5085 := [[435.72, -21.72, 181.07], [-0.035816, 0.706199, 0.704887, 0.055981], [0,0,0,0], [9E9, 9E9, 9E9, 9E9, 9E9, 9E9]];
	VAR robtarget Openhole_5086 := [[436.14, -21.45, 181.11], [-0.035315, 0.706224, 0.705066, 0.053688], [0,0,0,0], [9E9, 9E9, 9E9, 9E9, 9E9, 9E9]];
	VAR robtarget Openhole_5087 := [[436.96, -20.89, 181.2], [-0.034451, 0.706267, 0.705403, 0.049062], [0,0,0,0], [9E9, 9E9, 9E9, 9E9, 9E9, 9E9]];
	VAR robtarget Openhole_5088 := [[437.76, -20.3, 181.28], [-0.033756, 0.706301, 0.705712, 0.044393], [0,0,0,0], [9E9, 9E9, 9E9, 9E9, 9E9, 9E9]];
	VAR robtarget Openhole_5089 := [[438.17, -20.01, 181.32], [-0.033349, 0.70632, 0.705855, 0.042063], [0,0,0,0], [9E9, 9E9, 9E9, 9E9, 9E9, 9E9]];
	VAR robtarget Openhole_5090 := [[441.8, -21.35, 181.25], [-0.016527, 0.706914, 0.70627, 0.034399], [0,0,0,0], [9E9, 9E9, 9E9, 9E9, 9E9, 9E9]];
	VAR robtarget Openhole_5091 := [[441.01, -21.74, 181.2], [-0.017882, 0.706881, 0.706064, 0.038379], [0,0,0,0], [9E9, 9E9, 9E9, 9E9, 9E9, 9E9]];
	VAR robtarget Openhole_5092 := [[440.59, -22.01, 181.17], [-0.018391, 0.706868, 0.705935, 0.0407], [0,0,0,0], [9E9, 9E9, 9E9, 9E9, 9E9, 9E9]];
	VAR robtarget Openhole_5093 := [[439.34, -22.84, 181.05], [-0.019808, 0.706829, 0.705498, 0.047665], [0,0,0,0], [9E9, 9E9, 9E9, 9E9, 9E9, 9E9]];
	VAR robtarget Openhole_5094 := [[438.06, -23.61, 180.92], [-0.021521, 0.706779, 0.705001, 0.054533], [0,0,0,0], [9E9, 9E9, 9E9, 9E9, 9E9, 9E9]];
	VAR robtarget Openhole_5095 := [[437.63, -23.85, 180.88], [-0.022197, 0.706758, 0.704823, 0.056786], [0,0,0,0], [9E9, 9E9, 9E9, 9E9, 9E9, 9E9]];
	VAR robtarget Openhole_5096 := [[435.85, -24.75, 180.68], [-0.025165, 0.706659, 0.70405, 0.065677], [0,0,0,0], [9E9, 9E9, 9E9, 9E9, 9E9, 9E9]];
	VAR robtarget Openhole_5097 := [[432.92, -27.42, 180.1], [-0.026084, 0.706626, 0.702083, 0.084136], [0,0,0,0], [9E9, 9E9, 9E9, 9E9, 9E9, 9E9]];
	VAR robtarget Openhole_5098 := [[434.35, -26.98, 180.27], [-0.022739, 0.706741, 0.702786, 0.078054], [0,0,0,0], [9E9, 9E9, 9E9, 9E9, 9E9, 9E9]];
	VAR robtarget Openhole_5099 := [[438.55, -25.44, 180.75], [-0.013695, 0.706974, 0.704635, 0.059067], [0,0,0,0], [9E9, 9E9, 9E9, 9E9, 9E9, 9E9]];
	VAR robtarget Openhole_5100 := [[439.46, -25.04, 180.85], [-0.011955, 0.707006, 0.704989, 0.054687], [0,0,0,0], [9E9, 9E9, 9E9, 9E9, 9E9, 9E9]];
	VAR robtarget Openhole_5101 := [[439.91, -24.83, 180.89], [-0.011132, 0.707019, 0.705157, 0.052473], [0,0,0,0], [9E9, 9E9, 9E9, 9E9, 9E9, 9E9]];
	VAR robtarget Openhole_5102 := [[440.8, -24.39, 180.98], [-0.009596, 0.707042, 0.705476, 0.047998], [0,0,0,0], [9E9, 9E9, 9E9, 9E9, 9E9, 9E9]];
	VAR robtarget Openhole_5103 := [[441.23, -24.14, 181.02], [-0.008983, 0.70705, 0.705628, 0.045709], [0,0,0,0], [9E9, 9E9, 9E9, 9E9, 9E9, 9E9]];
	VAR robtarget Openhole_5104 := [[441.65, -23.86, 181.06], [-0.008494, 0.707056, 0.705774, 0.043388], [0,0,0,0], [9E9, 9E9, 9E9, 9E9, 9E9, 9E9]];
	VAR robtarget Openhole_5105 := [[442.05, -23.57, 181.1], [-0.008109, 0.70706, 0.705915, 0.041045], [0,0,0,0], [9E9, 9E9, 9E9, 9E9, 9E9, 9E9]];
	VAR robtarget Openhole_5106 := [[442.67, -23.11, 181.16], [-0.007581, 0.707066, 0.706117, 0.037409], [0,0,0,0], [9E9, 9E9, 9E9, 9E9, 9E9, 9E9]];
	VAR robtarget Openhole_5107 := [[445.06, -25.46, 181.16], [0.008554, 0.707055, 0.706124, 0.03727], [0,0,0,0], [9E9, 9E9, 9E9, 9E9, 9E9, 9E9]];
	VAR robtarget Openhole_5108 := [[444.46, -25.91, 181.1], [0.008023, 0.707061, 0.705925, 0.040863], [0,0,0,0], [9E9, 9E9, 9E9, 9E9, 9E9, 9E9]];
	VAR robtarget Openhole_5109 := [[443.53, -26.29, 181.01], [0.006171, 0.70708, 0.705658, 0.045248], [0,0,0,0], [9E9, 9E9, 9E9, 9E9, 9E9, 9E9]];
	VAR robtarget Openhole_5110 := [[443.06, -26.45, 180.97], [0.005086, 0.707088, 0.705519, 0.047365], [0,0,0,0], [9E9, 9E9, 9E9, 9E9, 9E9, 9E9]];
	VAR robtarget Openhole_5111 := [[442.11, -26.73, 180.88], [0.002768, 0.707101, 0.705228, 0.051513], [0,0,0,0], [9E9, 9E9, 9E9, 9E9, 9E9, 9E9]];
	VAR robtarget Openhole_5112 := [[441.62, -26.84, 180.84], [0.001476, 0.707105, 0.70508, 0.053506], [0,0,0,0], [9E9, 9E9, 9E9, 9E9, 9E9, 9E9]];
	VAR robtarget Openhole_5113 := [[437.75, -27.77, 180.45], [-0.008546, 0.707055, 0.703682, 0.06951], [0,0,0,0], [9E9, 9E9, 9E9, 9E9, 9E9, 9E9]];
	VAR robtarget Openhole_5114 := [[431.47, -29.27, 179.66], [-0.024783, 0.706672, 0.700706, 0.094929], [0,0,0,0], [9E9, 9E9, 9E9, 9E9, 9E9, 9E9]];
	VAR robtarget Openhole_5115 := [[428.05, -31.34, 178.9], [-0.02942, 0.706494, 0.698092, 0.112548], [0,0,0,0], [9E9, 9E9, 9E9, 9E9, 9E9, 9E9]];
	VAR robtarget Openhole_5116 := [[437.85, -29.84, 180.23], [-0.001273, 0.707106, 0.703005, 0.076049], [0,0,0,0], [9E9, 9E9, 9E9, 9E9, 9E9, 9E9]];
	VAR robtarget Openhole_5117 := [[439.82, -29.61, 180.45], [0.004674, 0.707091, 0.703757, 0.068746], [0,0,0,0], [9E9, 9E9, 9E9, 9E9, 9E9, 9E9]];
	VAR robtarget Openhole_5118 := [[441.81, -29.49, 180.66], [0.01106, 0.70702, 0.704406, 0.061745], [0,0,0,0], [9E9, 9E9, 9E9, 9E9, 9E9, 9E9]];
	VAR robtarget Openhole_5119 := [[443.3, -29.47, 180.81], [0.016081, 0.706924, 0.704832, 0.056676], [0,0,0,0], [9E9, 9E9, 9E9, 9E9, 9E9, 9E9]];
	VAR robtarget Openhole_5120 := [[450.76, -29.75, 181.57], [0.042447, 0.705832, 0.706363, 0.03243], [0,0,0,0], [9E9, 9E9, 9E9, 9E9, 9E9, 9E9]];
	VAR robtarget Openhole_5121 := [[451.25, -29.75, 181.62], [0.044139, 0.705728, 0.706438, 0.030742], [0,0,0,0], [9E9, 9E9, 9E9, 9E9, 9E9, 9E9]];
	VAR robtarget Openhole_5122 := [[451.75, -29.75, 181.67], [0.045814, 0.705621, 0.70651, 0.029042], [0,0,0,0], [9E9, 9E9, 9E9, 9E9, 9E9, 9E9]];
	VAR robtarget Openhole_5123 := [[455.72, -29.42, 182.06], [0.058124, 0.704714, 0.706959, 0.014459], [0,0,0,0], [9E9, 9E9, 9E9, 9E9, 9E9, 9E9]];
	VAR robtarget Openhole_5124 := [[458.68, -29.06, 182.32], [0.066825, 0.703942, 0.7071, 0.003138], [0,0,0,0], [9E9, 9E9, 9E9, 9E9, 9E9, 9E9]];
	VAR robtarget Openhole_5125 := [[468.12, -28.35, 183.11], [0.095382, 0.700644, 0.706422, -0.031123], [0,0,0,0], [9E9, 9E9, 9E9, 9E9, 9E9, 9E9]];
	VAR robtarget Openhole_5126 := [[481.57, -27.6, 184.08], [0.134584, 0.694181, 0.702858, -0.077402], [0,0,0,0], [9E9, 9E9, 9E9, 9E9, 9E9, 9E9]];
	VAR robtarget Openhole_5127 := [[483.56, -27.51, 184.22], [0.14018, 0.693072, 0.702105, -0.083955], [0,0,0,0], [9E9, 9E9, 9E9, 9E9, 9E9, 9E9]];
	VAR robtarget Openhole_5128 := [[481.55, -17.51, 180.95], [0.102219, 0.699679, 0.698535, -0.109767], [0,0,0,0], [9E9, 9E9, 9E9, 9E9, 9E9, 9E9]];
	VAR robtarget Openhole_5129 := [[491.04, -17.63, 180.86], [0.130963, 0.694873, 0.693601, -0.137539], [0,0,0,0], [9E9, 9E9, 9E9, 9E9, 9E9, 9E9]];
	VAR robtarget Openhole_5130 := [[491.54, -17.62, 180.85], [0.132401, 0.694601, 0.693316, -0.138972], [0,0,0,0], [9E9, 9E9, 9E9, 9E9, 9E9, 9E9]];
	VAR robtarget Openhole_5131 := [[500.54, -17.43, 180.64], [0.156815, 0.689499, 0.687747, -0.164329], [0,0,0,0], [9E9, 9E9, 9E9, 9E9, 9E9, 9E9]];
	VAR robtarget Openhole_5132 := [[503.53, -17.27, 180.51], [0.164262, 0.687763, 0.68571, -0.172632], [0,0,0,0], [9E9, 9E9, 9E9, 9E9, 9E9, 9E9]];
	VAR robtarget Openhole_5133 := [[504.34, -17.24, 180.48], [0.166288, 0.687276, 0.685158, -0.174811], [0,0,0,0], [9E9, 9E9, 9E9, 9E9, 9E9, 9E9]];
	VAR robtarget Openhole_5134 := [[509.34, -17.24, 180.39], [0.183051, 0.683002, 0.683002, -0.183051], [0,0,0,0], [9E9, 9E9, 9E9, 9E9, 9E9, 9E9]];
	VAR robtarget Openhole_5135 := [[536.34, -17.24, 180.3], [0.183051, 0.683002, 0.683002, -0.183051], [0,0,0,0], [9E9, 9E9, 9E9, 9E9, 9E9, 9E9]];
	VAR robtarget Openhole_5136 := [[536.34, -17.96, 180.72], [0.183051, 0.683002, 0.683002, -0.183051], [0,0,0,0], [9E9, 9E9, 9E9, 9E9, 9E9, 9E9]];
	VAR robtarget Openhole_5137 := [[509.34, -17.96, 180.81], [0.183051, 0.683002, 0.683002, -0.183051], [0,0,0,0], [9E9, 9E9, 9E9, 9E9, 9E9, 9E9]];
	VAR robtarget Openhole_5138 := [[504.35, -17.96, 180.86], [0.168399, 0.686762, 0.68569, -0.17271], [0,0,0,0], [9E9, 9E9, 9E9, 9E9, 9E9, 9E9]];
	VAR robtarget Openhole_5139 := [[496.08, -18.29, 181.09], [0.147265, 0.691602, 0.691081, -0.149689], [0,0,0,0], [9E9, 9E9, 9E9, 9E9, 9E9, 9E9]];
	VAR robtarget Openhole_5140 := [[491.09, -18.34, 181.15], [0.133298, 0.694429, 0.694013, -0.135447], [0,0,0,0], [9E9, 9E9, 9E9, 9E9, 9E9, 9E9]];
	VAR robtarget Openhole_5141 := [[490.59, -18.34, 181.15], [0.131855, 0.694704, 0.694292, -0.134009], [0,0,0,0], [9E9, 9E9, 9E9, 9E9, 9E9, 9E9]];
	VAR robtarget Openhole_5142 := [[474.59, -18.11, 181.2], [0.082342, 0.702296, 0.701848, -0.086076], [0,0,0,0], [9E9, 9E9, 9E9, 9E9, 9E9, 9E9]];
	VAR robtarget Openhole_5143 := [[474.09, -18.11, 181.2], [0.080746, 0.702481, 0.702042, -0.084479], [0,0,0,0], [9E9, 9E9, 9E9, 9E9, 9E9, 9E9]];
	VAR robtarget Openhole_5144 := [[471.09, -18.16, 181.24], [0.071228, 0.70351, 0.703152, -0.074678], [0,0,0,0], [9E9, 9E9, 9E9, 9E9, 9E9, 9E9]];
	VAR robtarget Openhole_5145 := [[469.59, -18.24, 181.27], [0.066606, 0.703963, 0.703677, -0.069558], [0,0,0,0], [9E9, 9E9, 9E9, 9E9, 9E9, 9E9]];
	VAR robtarget Openhole_5146 := [[467.1, -18.42, 181.32], [0.059024, 0.704639, 0.704488, -0.060795], [0,0,0,0], [9E9, 9E9, 9E9, 9E9, 9E9, 9E9]];
	VAR robtarget Openhole_5147 := [[466.6, -18.47, 181.33], [0.057575, 0.704759, 0.704644, -0.058969], [0,0,0,0], [9E9, 9E9, 9E9, 9E9, 9E9, 9E9]];
	VAR robtarget Openhole_5148 := [[467.28, -16.77, 181.03], [0.054116, 0.705033, 0.703935, -0.066896], [0,0,0,0], [9E9, 9E9, 9E9, 9E9, 9E9, 9E9]];
	VAR robtarget Openhole_5149 := [[468.25, -16.53, 180.97], [0.056526, 0.704844, 0.703548, -0.070855], [0,0,0,0], [9E9, 9E9, 9E9, 9E9, 9E9, 9E9]];
	VAR robtarget Openhole_5150 := [[469.23, -16.32, 180.9], [0.059025, 0.704639, 0.703146, -0.074737], [0,0,0,0], [9E9, 9E9, 9E9, 9E9, 9E9, 9E9]];
	VAR robtarget Openhole_5151 := [[469.72, -16.22, 180.87], [0.060313, 0.70453, 0.702941, -0.076645], [0,0,0,0], [9E9, 9E9, 9E9, 9E9, 9E9, 9E9]];
	VAR robtarget Openhole_5152 := [[470.21, -16.14, 180.84], [0.061637, 0.704415, 0.702733, -0.078522], [0,0,0,0], [9E9, 9E9, 9E9, 9E9, 9E9, 9E9]];
	VAR robtarget Openhole_5153 := [[472.19, -15.88, 180.73], [0.067235, 0.703903, 0.701888, -0.085751], [0,0,0,0], [9E9, 9E9, 9E9, 9E9, 9E9, 9E9]];
	VAR robtarget Openhole_5154 := [[473.18, -15.79, 180.68], [0.070173, 0.703616, 0.701456, -0.089216], [0,0,0,0], [9E9, 9E9, 9E9, 9E9, 9E9, 9E9]];
	VAR robtarget Openhole_5155 := [[478.67, -15.58, 180.45], [0.087044, 0.701729, 0.698945, -0.107125], [0,0,0,0], [9E9, 9E9, 9E9, 9E9, 9E9, 9E9]];
	VAR robtarget Openhole_5156 := [[479.17, -15.58, 180.43], [0.088614, 0.701532, 0.698706, -0.10867], [0,0,0,0], [9E9, 9E9, 9E9, 9E9, 9E9, 9E9]];
	VAR robtarget Openhole_5157 := [[479.67, -15.58, 180.42], [0.090185, 0.701332, 0.698466, -0.110206], [0,0,0,0], [9E9, 9E9, 9E9, 9E9, 9E9, 9E9]];
	VAR robtarget Openhole_5158 := [[492.67, -15.73, 180.05], [0.129772, 0.695097, 0.69145, -0.147976], [0,0,0,0], [9E9, 9E9, 9E9, 9E9, 9E9, 9E9]];
	VAR robtarget Openhole_5159 := [[493.16, -15.73, 180.03], [0.131204, 0.694828, 0.691148, -0.149379], [0,0,0,0], [9E9, 9E9, 9E9, 9E9, 9E9, 9E9]];
	VAR robtarget Openhole_5160 := [[500.66, -15.57, 179.71], [0.151584, 0.690668, 0.686328, -0.170158], [0,0,0,0], [9E9, 9E9, 9E9, 9E9, 9E9, 9E9]];
	VAR robtarget Openhole_5161 := [[503.64, -15.39, 179.52], [0.159031, 0.688991, 0.684227, -0.178419], [0,0,0,0], [9E9, 9E9, 9E9, 9E9, 9E9, 9E9]];
	VAR robtarget Openhole_5162 := [[504.34, -15.36, 179.48], [0.160771, 0.688587, 0.683738, -0.180284], [0,0,0,0], [9E9, 9E9, 9E9, 9E9, 9E9, 9E9]];
	VAR robtarget Openhole_5163 := [[509.34, -15.36, 179.3], [0.183051, 0.683002, 0.683002, -0.183051], [0,0,0,0], [9E9, 9E9, 9E9, 9E9, 9E9, 9E9]];
	VAR robtarget Openhole_5164 := [[536.34, -15.36, 179.22], [0.183051, 0.683002, 0.683002, -0.183051], [0,0,0,0], [9E9, 9E9, 9E9, 9E9, 9E9, 9E9]];
	VAR robtarget Openhole_5165 := [[536.34, -14.15, 178.52], [0.183051, 0.683002, 0.683002, -0.183051], [0,0,0,0], [9E9, 9E9, 9E9, 9E9, 9E9, 9E9]];
	VAR robtarget Openhole_5166 := [[509.34, -14.15, 178.6], [0.183051, 0.683002, 0.683002, -0.183051], [0,0,0,0], [9E9, 9E9, 9E9, 9E9, 9E9, 9E9]];
	VAR robtarget Openhole_5167 := [[504.34, -14.15, 178.84], [0.157228, 0.689405, 0.682805, -0.183787], [0,0,0,0], [9E9, 9E9, 9E9, 9E9, 9E9, 9E9]];
	VAR robtarget Openhole_5168 := [[498.3, -14.46, 179.27], [0.141803, 0.692742, 0.68705, -0.16722], [0,0,0,0], [9E9, 9E9, 9E9, 9E9, 9E9, 9E9]];
	VAR robtarget Openhole_5169 := [[493.8, -14.52, 179.49], [0.129301, 0.695184, 0.689942, -0.154854], [0,0,0,0], [9E9, 9E9, 9E9, 9E9, 9E9, 9E9]];
	VAR robtarget Openhole_5170 := [[493.3, -14.52, 179.51], [0.127863, 0.69545, 0.690251, -0.153473], [0,0,0,0], [9E9, 9E9, 9E9, 9E9, 9E9, 9E9]];
	VAR robtarget Openhole_5171 := [[480.81, -14.37, 180.01], [0.08985, 0.701375, 0.697262, -0.117581], [0,0,0,0], [9E9, 9E9, 9E9, 9E9, 9E9, 9E9]];
	VAR robtarget Openhole_5172 := [[480.31, -14.37, 180.03], [0.088294, 0.701573, 0.697518, -0.116054], [0,0,0,0], [9E9, 9E9, 9E9, 9E9, 9E9, 9E9]];
	VAR robtarget Openhole_5173 := [[475.32, -14.53, 180.3], [0.072937, 0.703335, 0.699983, -0.10012], [0,0,0,0], [9E9, 9E9, 9E9, 9E9, 9E9, 9E9]];
	VAR robtarget Openhole_5174 := [[472.35, -14.82, 180.49], [0.064258, 0.704181, 0.70139, -0.089731], [0,0,0,0], [9E9, 9E9, 9E9, 9E9, 9E9, 9E9]];
	VAR robtarget Openhole_5175 := [[471.85, -14.89, 180.53], [0.062882, 0.704305, 0.701619, -0.087922], [0,0,0,0], [9E9, 9E9, 9E9, 9E9, 9E9, 9E9]];
	VAR robtarget Openhole_5176 := [[471.36, -14.97, 180.56], [0.061542, 0.704424, 0.701848, -0.08608], [0,0,0,0], [9E9, 9E9, 9E9, 9E9, 9E9, 9E9]];
	VAR robtarget Openhole_5177 := [[469.41, -15.37, 180.72], [0.056462, 0.704849, 0.70274, -0.078461], [0,0,0,0], [9E9, 9E9, 9E9, 9E9, 9E9, 9E9]];
	VAR robtarget Openhole_5178 := [[468.44, -15.62, 180.8], [0.054118, 0.705033, 0.703172, -0.074497], [0,0,0,0], [9E9, 9E9, 9E9, 9E9, 9E9, 9E9]];
	VAR robtarget Openhole_5179 := [[467.01, -16.05, 180.92], [0.050803, 0.705279, 0.703791, -0.068398], [0,0,0,0], [9E9, 9E9, 9E9, 9E9, 9E9, 9E9]];
	VAR robtarget Openhole_5180 := [[466.54, -16.21, 180.96], [0.0498, 0.705351, 0.703991, -0.066305], [0,0,0,0], [9E9, 9E9, 9E9, 9E9, 9E9, 9E9]];
	VAR robtarget Openhole_5181 := [[465.61, -16.58, 181.04], [0.047929, 0.705481, 0.70438, -0.062041], [0,0,0,0], [9E9, 9E9, 9E9, 9E9, 9E9, 9E9]];
	VAR robtarget Openhole_5182 := [[465.15, -16.77, 181.08], [0.047037, 0.705541, 0.704566, -0.059884], [0,0,0,0], [9E9, 9E9, 9E9, 9E9, 9E9, 9E9]];
	VAR robtarget Openhole_5183 := [[463.78, -17.37, 181.19], [0.044524, 0.705704, 0.705094, -0.053321], [0,0,0,0], [9E9, 9E9, 9E9, 9E9, 9E9, 9E9]];
	VAR robtarget Openhole_5184 := [[462.86, -17.76, 181.26], [0.042757, 0.705813, 0.70541, -0.04896], [0,0,0,0], [9E9, 9E9, 9E9, 9E9, 9E9, 9E9]];
	VAR robtarget Openhole_5185 := [[462.42, -18, 181.29], [0.042075, 0.705854, 0.705563, -0.046703], [0,0,0,0], [9E9, 9E9, 9E9, 9E9, 9E9, 9E9]];
	VAR robtarget Openhole_5186 := [[461.97, -18.21, 181.32], [0.041269, 0.705901, 0.705706, -0.044484], [0,0,0,0], [9E9, 9E9, 9E9, 9E9, 9E9, 9E9]];
	VAR robtarget Openhole_5187 := [[462.15, -19.58, 181.49], [0.046479, 0.705578, 0.705948, -0.040461], [0,0,0,0], [9E9, 9E9, 9E9, 9E9, 9E9, 9E9]];
	VAR robtarget Openhole_5188 := [[462.64, -19.54, 181.49], [0.048003, 0.705475, 0.705842, -0.042267], [0,0,0,0], [9E9, 9E9, 9E9, 9E9, 9E9, 9E9]];
	VAR robtarget Openhole_5189 := [[463.64, -19.43, 181.48], [0.050964, 0.705268, 0.705613, -0.04594], [0,0,0,0], [9E9, 9E9, 9E9, 9E9, 9E9, 9E9]];
	VAR robtarget Openhole_5190 := [[464.14, -19.42, 181.48], [0.052604, 0.705147, 0.705501, -0.04763], [0,0,0,0], [9E9, 9E9, 9E9, 9E9, 9E9, 9E9]];
	VAR robtarget Openhole_5191 := [[464.64, -19.38, 181.47], [0.054126, 0.705032, 0.705378, -0.04942], [0,0,0,0], [9E9, 9E9, 9E9, 9E9, 9E9, 9E9]];
	VAR robtarget Openhole_5192 := [[465.64, -19.33, 181.47], [0.05725, 0.704785, 0.705124, -0.052918], [0,0,0,0], [9E9, 9E9, 9E9, 9E9, 9E9, 9E9]];
	VAR robtarget Openhole_5193 := [[466.14, -19.31, 181.47], [0.058851, 0.704654, 0.704994, -0.054623], [0,0,0,0], [9E9, 9E9, 9E9, 9E9, 9E9, 9E9]];
	VAR robtarget Openhole_5194 := [[466.64, -19.31, 181.47], [0.060488, 0.704515, 0.704863, -0.056288], [0,0,0,0], [9E9, 9E9, 9E9, 9E9, 9E9, 9E9]];
	VAR robtarget Openhole_5195 := [[469.13, -19.24, 181.46], [0.068449, 0.703786, 0.704137, -0.064741], [0,0,0,0], [9E9, 9E9, 9E9, 9E9, 9E9, 9E9]];
	VAR robtarget Openhole_5196 := [[469.63, -19.24, 181.46], [0.070088, 0.703625, 0.703985, -0.066368], [0,0,0,0], [9E9, 9E9, 9E9, 9E9, 9E9, 9E9]];
	VAR robtarget Openhole_5197 := [[470.13, -19.24, 181.46], [0.071713, 0.703461, 0.703829, -0.068001], [0,0,0,0], [9E9, 9E9, 9E9, 9E9, 9E9, 9E9]];
	VAR robtarget Openhole_5198 := [[470.63, -19.24, 181.47], [0.073339, 0.703293, 0.70367, -0.069627], [0,0,0,0], [9E9, 9E9, 9E9, 9E9, 9E9, 9E9]];
	VAR robtarget Openhole_5199 := [[490.13, -19.56, 181.63], [0.134326, 0.694231, 0.695258, -0.128906], [0,0,0,0], [9E9, 9E9, 9E9, 9E9, 9E9, 9E9]];
	VAR robtarget Openhole_5200 := [[490.63, -19.56, 181.63], [0.135764, 0.693951, 0.694987, -0.130359], [0,0,0,0], [9E9, 9E9, 9E9, 9E9, 9E9, 9E9]];
	VAR robtarget Openhole_5201 := [[499.63, -19.4, 181.6], [0.160237, 0.688712, 0.689675, -0.156038], [0,0,0,0], [9E9, 9E9, 9E9, 9E9, 9E9, 9E9]];
	VAR robtarget Openhole_5202 := [[504.35, -19.19, 181.51], [0.171977, 0.685875, 0.686579, -0.169145], [0,0,0,0], [9E9, 9E9, 9E9, 9E9, 9E9, 9E9]];
	VAR robtarget Openhole_5203 := [[536.35, -19.19, 181.43], [0.183051, 0.683002, 0.683002, -0.183051], [0,0,0,0], [9E9, 9E9, 9E9, 9E9, 9E9, 9E9]];
	VAR robtarget Openhole_5204 := [[536.35, -19.88, 181.83], [0.183051, 0.683002, 0.683002, -0.183051], [0,0,0,0], [9E9, 9E9, 9E9, 9E9, 9E9, 9E9]];
	VAR robtarget Openhole_5205 := [[509.35, -19.88, 181.92], [0.183051, 0.683002, 0.683002, -0.183051], [0,0,0,0], [9E9, 9E9, 9E9, 9E9, 9E9, 9E9]];
	VAR robtarget Openhole_5206 := [[504.35, -19.88, 181.88], [0.174012, 0.685361, 0.687076, -0.167111], [0,0,0,0], [9E9, 9E9, 9E9, 9E9, 9E9, 9E9]];
	VAR robtarget Openhole_5207 := [[495.85, -20.21, 181.95], [0.152427, 0.690482, 0.692451, -0.143218], [0,0,0,0], [9E9, 9E9, 9E9, 9E9, 9E9, 9E9]];
	VAR robtarget Openhole_5208 := [[489.35, -20.27, 181.9], [0.134298, 0.694236, 0.696079, -0.124397], [0,0,0,0], [9E9, 9E9, 9E9, 9E9, 9E9, 9E9]];
	VAR robtarget Openhole_5209 := [[488.85, -20.27, 181.89], [0.132849, 0.694515, 0.696339, -0.122928], [0,0,0,0], [9E9, 9E9, 9E9, 9E9, 9E9, 9E9]];
	VAR robtarget Openhole_5210 := [[474.85, -20.03, 181.67], [0.089502, 0.70142, 0.702496, -0.080622], [0,0,0,0], [9E9, 9E9, 9E9, 9E9, 9E9, 9E9]];
	VAR robtarget Openhole_5211 := [[470.86, -19.93, 181.61], [0.076344, 0.702973, 0.703823, -0.068065], [0,0,0,0], [9E9, 9E9, 9E9, 9E9, 9E9, 9E9]];
	VAR robtarget Openhole_5212 := [[473.3, -13.93, 180.25], [0.064444, 0.704164, 0.700602, -0.095694], [0,0,0,0], [9E9, 9E9, 9E9, 9E9, 9E9, 9E9]];
	VAR robtarget Openhole_5213 := [[474.29, -13.82, 180.17], [0.067296, 0.703897, 0.700116, -0.099186], [0,0,0,0], [9E9, 9E9, 9E9, 9E9, 9E9, 9E9]];
	VAR robtarget Openhole_5214 := [[479.28, -13.55, 179.84], [0.082366, 0.702293, 0.697606, -0.115523], [0,0,0,0], [9E9, 9E9, 9E9, 9E9, 9E9, 9E9]];
	VAR robtarget Openhole_5215 := [[482.27, -13.53, 179.68], [0.091677, 0.701139, 0.696028, -0.12468], [0,0,0,0], [9E9, 9E9, 9E9, 9E9, 9E9, 9E9]];
	VAR robtarget Openhole_5216 := [[482.77, -13.53, 179.65], [0.093236, 0.700933, 0.69576, -0.126168], [0,0,0,0], [9E9, 9E9, 9E9, 9E9, 9E9, 9E9]];
	VAR robtarget Openhole_5217 := [[494.76, -13.69, 179.09], [0.129496, 0.695148, 0.688769, -0.159991], [0,0,0,0], [9E9, 9E9, 9E9, 9E9, 9E9, 9E9]];
	VAR robtarget Openhole_5218 := [[495.26, -13.69, 179.06], [0.130919, 0.694881, 0.688451, -0.161355], [0,0,0,0], [9E9, 9E9, 9E9, 9E9, 9E9, 9E9]];
	VAR robtarget Openhole_5219 := [[501.74, -13.52, 178.64], [0.148419, 0.691355, 0.684072, -0.179011], [0,0,0,0], [9E9, 9E9, 9E9, 9E9, 9E9, 9E9]];
	VAR robtarget Openhole_5220 := [[504.34, -13.35, 178.41], [0.154882, 0.689936, 0.682177, -0.186102], [0,0,0,0], [9E9, 9E9, 9E9, 9E9, 9E9, 9E9]];
	VAR robtarget Openhole_5221 := [[509.34, -13.35, 178.14], [0.183051, 0.683002, 0.683002, -0.183051], [0,0,0,0], [9E9, 9E9, 9E9, 9E9, 9E9, 9E9]];
	VAR robtarget Openhole_5222 := [[536.34, -13.35, 178.06], [0.183051, 0.683002, 0.683002, -0.183051], [0,0,0,0], [9E9, 9E9, 9E9, 9E9, 9E9, 9E9]];
	VAR robtarget Openhole_5223 := [[536.33, -11.35, 176.9], [0.183051, 0.683002, 0.683002, -0.183051], [0,0,0,0], [9E9, 9E9, 9E9, 9E9, 9E9, 9E9]];
	VAR robtarget Openhole_5224 := [[509.33, -11.35, 176.99], [0.183051, 0.683002, 0.683002, -0.183051], [0,0,0,0], [9E9, 9E9, 9E9, 9E9, 9E9, 9E9]];
	VAR robtarget Openhole_5225 := [[504.33, -11.35, 177.36], [0.149024, 0.691225, 0.680579, -0.191864], [0,0,0,0], [9E9, 9E9, 9E9, 9E9, 9E9, 9E9]];
	VAR robtarget Openhole_5226 := [[503.51, -11.37, 177.43], [0.14689, 0.691681, 0.681171, -0.189753], [0,0,0,0], [9E9, 9E9, 9E9, 9E9, 9E9, 9E9]];
	VAR robtarget Openhole_5227 := [[498.54, -11.56, 177.89], [0.133766, 0.694339, 0.68473, -0.176479], [0,0,0,0], [9E9, 9E9, 9E9, 9E9, 9E9, 9E9]];
	VAR robtarget Openhole_5228 := [[497.54, -11.57, 177.96], [0.130974, 0.694871, 0.685404, -0.173843], [0,0,0,0], [9E9, 9E9, 9E9, 9E9, 9E9, 9E9]];
	VAR robtarget Openhole_5229 := [[497.04, -11.57, 178], [0.129556, 0.695137, 0.685736, -0.172528], [0,0,0,0], [9E9, 9E9, 9E9, 9E9, 9E9, 9E9]];
	VAR robtarget Openhole_5230 := [[482.58, -11.27, 178.94], [0.085403, 0.70193, 0.694533, -0.132753], [0,0,0,0], [9E9, 9E9, 9E9, 9E9, 9E9, 9E9]];
	VAR robtarget Openhole_5231 := [[482.08, -11.28, 178.98], [0.083847, 0.702118, 0.694816, -0.131264], [0,0,0,0], [9E9, 9E9, 9E9, 9E9, 9E9, 9E9]];
	VAR robtarget Openhole_5232 := [[477.1, -11.44, 179.39], [0.068544, 0.703777, 0.697583, -0.115664], [0,0,0,0], [9E9, 9E9, 9E9, 9E9, 9E9, 9E9]];
	VAR robtarget Openhole_5233 := [[473.15, -11.89, 179.79], [0.057205, 0.704789, 0.69973, -0.101872], [0,0,0,0], [9E9, 9E9, 9E9, 9E9, 9E9, 9E9]];
	VAR robtarget Openhole_5234 := [[471.68, -12.15, 179.94], [0.053239, 0.7051, 0.700508, -0.096377], [0,0,0,0], [9E9, 9E9, 9E9, 9E9, 9E9, 9E9]];
	VAR robtarget Openhole_5235 := [[471.19, -12.25, 180], [0.051975, 0.705194, 0.700765, -0.094493], [0,0,0,0], [9E9, 9E9, 9E9, 9E9, 9E9, 9E9]];
	VAR robtarget Openhole_5236 := [[470.71, -12.36, 180.05], [0.05075, 0.705283, 0.70102, -0.09258], [0,0,0,0], [9E9, 9E9, 9E9, 9E9, 9E9, 9E9]];
	VAR robtarget Openhole_5237 := [[469.27, -12.75, 180.22], [0.04728, 0.705524, 0.701773, -0.086684], [0,0,0,0], [9E9, 9E9, 9E9, 9E9, 9E9, 9E9]];
	VAR robtarget Openhole_5238 := [[468.32, -13.04, 180.33], [0.045099, 0.705667, 0.70226, -0.082652], [0,0,0,0], [9E9, 9E9, 9E9, 9E9, 9E9, 9E9]];
	VAR robtarget Openhole_5239 := [[467.85, -13.2, 180.38], [0.044061, 0.705733, 0.702498, -0.080602], [0,0,0,0], [9E9, 9E9, 9E9, 9E9, 9E9, 9E9]];
	VAR robtarget Openhole_5240 := [[467.38, -13.37, 180.44], [0.043082, 0.705793, 0.702734, -0.078518], [0,0,0,0], [9E9, 9E9, 9E9, 9E9, 9E9, 9E9]];
	VAR robtarget Openhole_5241 := [[466.46, -13.74, 180.55], [0.041245, 0.705903, 0.703194, -0.074282], [0,0,0,0], [9E9, 9E9, 9E9, 9E9, 9E9, 9E9]];
	VAR robtarget Openhole_5242 := [[466, -13.94, 180.61], [0.040397, 0.705952, 0.703418, -0.072128], [0,0,0,0], [9E9, 9E9, 9E9, 9E9, 9E9, 9E9]];
	VAR robtarget Openhole_5243 := [[465.55, -14.15, 180.66], [0.039593, 0.705997, 0.703638, -0.069952], [0,0,0,0], [9E9, 9E9, 9E9, 9E9, 9E9, 9E9]];
	VAR robtarget Openhole_5244 := [[464.66, -14.6, 180.77], [0.038128, 0.706078, 0.704063, -0.065539], [0,0,0,0], [9E9, 9E9, 9E9, 9E9, 9E9, 9E9]];
	VAR robtarget Openhole_5245 := [[463.8, -15.08, 180.87], [0.036849, 0.706146, 0.704466, -0.06105], [0,0,0,0], [9E9, 9E9, 9E9, 9E9, 9E9, 9E9]];
	VAR robtarget Openhole_5246 := [[462.94, -15.6, 180.97], [0.035726, 0.706204, 0.704846, -0.056503], [0,0,0,0], [9E9, 9E9, 9E9, 9E9, 9E9, 9E9]];
	VAR robtarget Openhole_5247 := [[462.52, -15.87, 181.02], [0.035223, 0.706229, 0.705026, -0.054209], [0,0,0,0], [9E9, 9E9, 9E9, 9E9, 9E9, 9E9]];
	VAR robtarget Openhole_5248 := [[460.89, -17, 181.2], [0.033558, 0.70631, 0.705678, -0.044928], [0,0,0,0], [9E9, 9E9, 9E9, 9E9, 9E9, 9E9]];
	VAR robtarget Openhole_5249 := [[461.06, -13.27, 180.77], [0.021544, 0.706779, 0.70472, -0.058048], [0,0,0,0], [9E9, 9E9, 9E9, 9E9, 9E9, 9E9]];
	VAR robtarget Openhole_5250 := [[460.62, -13.5, 180.82], [0.020835, 0.7068, 0.704901, -0.055805], [0,0,0,0], [9E9, 9E9, 9E9, 9E9, 9E9, 9E9]];
	VAR robtarget Openhole_5251 := [[458.51, -14.82, 181.05], [0.018118, 0.706875, 0.705717, -0.044311], [0,0,0,0], [9E9, 9E9, 9E9, 9E9, 9E9, 9E9]];
	VAR robtarget Openhole_5252 := [[457.68, -15.38, 181.13], [0.017233, 0.706897, 0.705994, -0.039648], [0,0,0,0], [9E9, 9E9, 9E9, 9E9, 9E9, 9E9]];
	VAR robtarget Openhole_5253 := [[456.81, -15.81, 181.19], [0.015719, 0.706932, 0.706228, -0.035235], [0,0,0,0], [9E9, 9E9, 9E9, 9E9, 9E9, 9E9]];
	VAR robtarget Openhole_5254 := [[457.02, -21.12, 181.58], [0.034484, 0.706265, 0.706878, -0.017973], [0,0,0,0], [9E9, 9E9, 9E9, 9E9, 9E9, 9E9]];
	VAR robtarget Openhole_5255 := [[463.93, -21.12, 181.72], [0.057616, 0.704756, 0.705905, -0.041207], [0,0,0,0], [9E9, 9E9, 9E9, 9E9, 9E9, 9E9]];
	VAR robtarget Openhole_5256 := [[469.41, -21.53, 181.91], [0.076975, 0.702905, 0.704724, -0.057995], [0,0,0,0], [9E9, 9E9, 9E9, 9E9, 9E9, 9E9]];
	VAR robtarget Openhole_5257 := [[482.39, -21.87, 182.32], [0.118792, 0.697057, 0.700229, -0.098386], [0,0,0,0], [9E9, 9E9, 9E9, 9E9, 9E9, 9E9]];
	VAR robtarget Openhole_5258 := [[487.39, -21.9, 182.47], [0.133699, 0.694352, 0.697939, -0.113498], [0,0,0,0], [9E9, 9E9, 9E9, 9E9, 9E9, 9E9]];
	VAR robtarget Openhole_5259 := [[487.89, -21.9, 182.49], [0.13515, 0.694071, 0.697694, -0.114993], [0,0,0,0], [9E9, 9E9, 9E9, 9E9, 9E9, 9E9]];
	VAR robtarget Openhole_5260 := [[498.39, -21.73, 182.7], [0.163904, 0.687848, 0.691944, -0.145649], [0,0,0,0], [9E9, 9E9, 9E9, 9E9, 9E9, 9E9]];
	VAR robtarget Openhole_5261 := [[503.38, -21.52, 182.72], [0.176334, 0.684767, 0.68882, -0.159773], [0,0,0,0], [9E9, 9E9, 9E9, 9E9, 9E9, 9E9]];
	VAR robtarget Openhole_5262 := [[504.35, -21.49, 182.73], [0.178705, 0.684153, 0.688202, -0.162413], [0,0,0,0], [9E9, 9E9, 9E9, 9E9, 9E9, 9E9]];
	VAR robtarget Openhole_5263 := [[509.35, -21.49, 182.85], [0.183051, 0.683002, 0.683002, -0.183051], [0,0,0,0], [9E9, 9E9, 9E9, 9E9, 9E9, 9E9]];
	VAR robtarget Openhole_5264 := [[536.24, -21.49, 182.76], [0.183051, 0.683002, 0.683002, -0.183051], [0,0,0,0], [9E9, 9E9, 9E9, 9E9, 9E9, 9E9]];
	VAR robtarget Openhole_5265 := [[536.33, -31.04, 188.28], [0.183051, 0.683002, 0.683002, -0.183051], [0,0,0,0], [9E9, 9E9, 9E9, 9E9, 9E9, 9E9]];
	VAR robtarget Openhole_5266 := [[509.37, -31.04, 188.36], [0.183051, 0.683002, 0.683002, -0.183051], [0,0,0,0], [9E9, 9E9, 9E9, 9E9, 9E9, 9E9]];
	VAR robtarget Openhole_5267 := [[504.38, -31.04, 187.78], [0.206267, 0.676353, 0.694185, -0.134564], [0,0,0,0], [9E9, 9E9, 9E9, 9E9, 9E9, 9E9]];
	VAR robtarget Openhole_5268 := [[486.98, -32.16, 186.18], [0.164388, 0.687733, 0.702572, -0.079951], [0,0,0,0], [9E9, 9E9, 9E9, 9E9, 9E9, 9E9]];
	VAR robtarget Openhole_5269 := [[478.56, -33.01, 185.35], [0.142761, 0.692546, 0.705309, -0.050384], [0,0,0,0], [9E9, 9E9, 9E9, 9E9, 9E9, 9E9]];
	VAR robtarget Openhole_5270 := [[471.68, -34.05, 184.65], [0.125145, 0.695944, 0.70669, -0.024262], [0,0,0,0], [9E9, 9E9, 9E9, 9E9, 9E9, 9E9]];
	VAR robtarget Openhole_5271 := [[465.83, -35.24, 183.99], [0.110593, 0.698405, 0.707106, -0.000646], [0,0,0,0], [9E9, 9E9, 9E9, 9E9, 9E9, 9E9]];
	VAR robtarget Openhole_5272 := [[458.15, -37.22, 182.96], [0.092036, 0.701092, 0.70638, 0.032045], [0,0,0,0], [9E9, 9E9, 9E9, 9E9, 9E9, 9E9]];
	VAR robtarget Openhole_5273 := [[452.92, -38.7, 182.1], [0.079446, 0.70263, 0.704986, 0.054724], [0,0,0,0], [9E9, 9E9, 9E9, 9E9, 9E9, 9E9]];
	VAR robtarget Openhole_5274 := [[457.28, -38.7, 182.92], [0.093939, 0.700839, 0.705983, 0.039847], [0,0,0,0], [9E9, 9E9, 9E9, 9E9, 9E9, 9E9]];
	VAR robtarget Openhole_5275 := [[457.75, -38.56, 183], [0.095092, 0.700684, 0.706097, 0.03778], [0,0,0,0], [9E9, 9E9, 9E9, 9E9, 9E9, 9E9]];
	VAR robtarget Openhole_5276 := [[466.4, -36.39, 184.27], [0.116112, 0.697508, 0.707106, 0.001196], [0,0,0,0], [9E9, 9E9, 9E9, 9E9, 9E9, 9E9]];
	VAR robtarget Openhole_5277 := [[473.19, -34.93, 185.07], [0.132656, 0.694552, 0.706611, -0.026476], [0,0,0,0], [9E9, 9E9, 9E9, 9E9, 9E9, 9E9]];
	VAR robtarget Openhole_5278 := [[479.58, -33.93, 185.76], [0.148652, 0.691305, 0.705282, -0.050768], [0,0,0,0], [9E9, 9E9, 9E9, 9E9, 9E9, 9E9]];
	VAR robtarget Openhole_5279 := [[487.99, -33.03, 186.63], [0.169854, 0.686404, 0.702524, -0.080372], [0,0,0,0], [9E9, 9E9, 9E9, 9E9, 9E9, 9E9]];
	VAR robtarget Openhole_5280 := [[504.38, -31.93, 188.25], [0.208768, 0.675586, 0.694682, -0.131975], [0,0,0,0], [9E9, 9E9, 9E9, 9E9, 9E9, 9E9]];
	VAR robtarget Openhole_5281 := [[509.37, -31.93, 188.87], [0.183051, 0.683002, 0.683002, -0.183051], [0,0,0,0], [9E9, 9E9, 9E9, 9E9, 9E9, 9E9]];
	VAR robtarget Openhole_5282 := [[536.37, -31.93, 188.79], [0.183051, 0.683002, 0.683002, -0.183051], [0,0,0,0], [9E9, 9E9, 9E9, 9E9, 9E9, 9E9]];
	VAR robtarget Openhole_5283 := [[536.37, -32.81, 189.3], [0.183051, 0.683002, 0.683002, -0.183051], [0,0,0,0], [9E9, 9E9, 9E9, 9E9, 9E9, 9E9]];
	VAR robtarget Openhole_5284 := [[524.37, -32.81, 189.33], [0.183051, 0.683002, 0.683002, -0.183051], [0,0,0,0], [9E9, 9E9, 9E9, 9E9, 9E9, 9E9]];
	VAR robtarget Openhole_5285 := [[509.37, -32.81, 189.38], [0.183051, 0.683002, 0.683002, -0.183051], [0,0,0,0], [9E9, 9E9, 9E9, 9E9, 9E9, 9E9]];
	VAR robtarget Openhole_5286 := [[504.38, -32.81, 188.72], [0.211268, 0.674808, 0.695167, -0.129396], [0,0,0,0], [9E9, 9E9, 9E9, 9E9, 9E9, 9E9]];
	VAR robtarget Openhole_5287 := [[488.99, -33.88, 187.09], [0.175191, 0.685061, 0.702468, -0.080865], [0,0,0,0], [9E9, 9E9, 9E9, 9E9, 9E9, 9E9]];
	VAR robtarget Openhole_5288 := [[481.09, -34.74, 186.22], [0.155585, 0.689778, 0.705111, -0.053084], [0,0,0,0], [9E9, 9E9, 9E9, 9E9, 9E9, 9E9]];
	VAR robtarget Openhole_5289 := [[474.71, -35.76, 185.5], [0.139878, 0.693133, 0.706517, -0.028866], [0,0,0,0], [9E9, 9E9, 9E9, 9E9, 9E9, 9E9]];
	VAR robtarget Openhole_5290 := [[467.43, -37.31, 184.6], [0.122335, 0.696444, 0.707106, 0.000684], [0,0,0,0], [9E9, 9E9, 9E9, 9E9, 9E9, 9E9]];
	VAR robtarget Openhole_5291 := [[462.62, -38.48, 183.9], [0.110705, 0.698387, 0.706799, 0.020876], [0,0,0,0], [9E9, 9E9, 9E9, 9E9, 9E9, 9E9]];
	VAR robtarget Openhole_5292 := [[462.13, -38.7, 183.84], [0.109821, 0.698527, 0.706726, 0.023208], [0,0,0,0], [9E9, 9E9, 9E9, 9E9, 9E9, 9E9]];
	VAR robtarget Openhole_5293 := [[466.52, -38.7, 184.67], [0.123836, 0.696179, 0.707059, 0.008225], [0,0,0,0], [9E9, 9E9, 9E9, 9E9, 9E9, 9E9]];
	VAR robtarget Openhole_5294 := [[467, -38.47, 184.72], [0.124686, 0.696027, 0.707082, 0.005886], [0,0,0,0], [9E9, 9E9, 9E9, 9E9, 9E9, 9E9]];
	VAR robtarget Openhole_5295 := [[474.26, -36.86, 185.7], [0.142024, 0.692697, 0.706706, -0.023813], [0,0,0,0], [9E9, 9E9, 9E9, 9E9, 9E9, 9E9]];
	VAR robtarget Openhole_5296 := [[481.12, -35.71, 186.52], [0.158697, 0.689068, 0.705331, -0.050082], [0,0,0,0], [9E9, 9E9, 9E9, 9E9, 9E9, 9E9]];
	VAR robtarget Openhole_5297 := [[489.01, -34.8, 187.44], [0.178021, 0.684331, 0.702785, -0.078061], [0,0,0,0], [9E9, 9E9, 9E9, 9E9, 9E9, 9E9]];
	VAR robtarget Openhole_5298 := [[501.89, -33.86, 188.92], [0.208287, 0.675734, 0.696963, -0.119341], [0,0,0,0], [9E9, 9E9, 9E9, 9E9, 9E9, 9E9]];
	VAR robtarget Openhole_5299 := [[504.38, -33.69, 189.19], [0.213761, 0.674022, 0.695641, -0.126819], [0,0,0,0], [9E9, 9E9, 9E9, 9E9, 9E9, 9E9]];
	VAR robtarget Openhole_5300 := [[509.37, -33.69, 189.89], [0.183051, 0.683002, 0.683002, -0.183051], [0,0,0,0], [9E9, 9E9, 9E9, 9E9, 9E9, 9E9]];
	VAR robtarget Openhole_5301 := [[536.37, -33.69, 189.81], [0.183051, 0.683002, 0.683002, -0.183051], [0,0,0,0], [9E9, 9E9, 9E9, 9E9, 9E9, 9E9]];
	VAR robtarget Openhole_5302 := [[536.38, -34.58, 190.32], [0.183051, 0.683002, 0.683002, -0.183051], [0,0,0,0], [9E9, 9E9, 9E9, 9E9, 9E9, 9E9]];
	VAR robtarget Openhole_5303 := [[509.38, -34.58, 190.4], [0.183051, 0.683002, 0.683002, -0.183051], [0,0,0,0], [9E9, 9E9, 9E9, 9E9, 9E9, 9E9]];
	VAR robtarget Openhole_5304 := [[504.37, -34.58, 189.65], [0.216241, 0.673231, 0.696107, -0.124239], [0,0,0,0], [9E9, 9E9, 9E9, 9E9, 9E9, 9E9]];
	VAR robtarget Openhole_5305 := [[490.51, -35.57, 187.97], [0.184366, 0.682649, 0.702528, -0.080342], [0,0,0,0], [9E9, 9E9, 9E9, 9E9, 9E9, 9E9]];
	VAR robtarget Openhole_5306 := [[482.13, -36.52, 186.94], [0.164071, 0.687809, 0.705277, -0.050831], [0,0,0,0], [9E9, 9E9, 9E9, 9E9, 9E9, 9E9]];
	VAR robtarget Openhole_5307 := [[475.27, -37.64, 186.06], [0.147513, 0.691549, 0.706675, -0.024704], [0,0,0,0], [9E9, 9E9, 9E9, 9E9, 9E9, 9E9]];
	VAR robtarget Openhole_5308 := [[470.91, -38.55, 185.47], [0.137115, 0.693686, 0.707071, -0.007112], [0,0,0,0], [9E9, 9E9, 9E9, 9E9, 9E9, 9E9]];
	VAR robtarget Openhole_5309 := [[470.42, -38.7, 185.41], [0.136036, 0.693898, 0.707089, -0.005054], [0,0,0,0], [9E9, 9E9, 9E9, 9E9, 9E9, 9E9]];
	VAR robtarget Openhole_5310 := [[474.82, -38.7, 186.24], [0.149416, 0.69114, 0.706827, -0.019872], [0,0,0,0], [9E9, 9E9, 9E9, 9E9, 9E9, 9E9]];
	VAR robtarget Openhole_5311 := [[475.31, -38.59, 186.31], [0.150571, 0.69089, 0.70677, -0.021807], [0,0,0,0], [9E9, 9E9, 9E9, 9E9, 9E9, 9E9]];
	VAR robtarget Openhole_5312 := [[482.64, -37.38, 187.3], [0.168181, 0.686815, 0.705351, -0.049798], [0,0,0,0], [9E9, 9E9, 9E9, 9E9, 9E9, 9E9]];
	VAR robtarget Openhole_5313 := [[491.02, -36.43, 188.4], [0.188254, 0.681587, 0.702646, -0.0793], [0,0,0,0], [9E9, 9E9, 9E9, 9E9, 9E9, 9E9]];
	VAR robtarget Openhole_5314 := [[502.39, -35.58, 189.87], [0.214387, 0.673824, 0.697576, -0.115704], [0,0,0,0], [9E9, 9E9, 9E9, 9E9, 9E9, 9E9]];
	VAR robtarget Openhole_5315 := [[504.37, -35.46, 190.12], [0.218719, 0.67243, 0.696561, -0.121669], [0,0,0,0], [9E9, 9E9, 9E9, 9E9, 9E9, 9E9]];
	VAR robtarget Openhole_5316 := [[504.37, -35.46, 190.12], [0.218724, 0.672428, 0.69656, -0.121675], [0,0,0,0], [9E9, 9E9, 9E9, 9E9, 9E9, 9E9]];
	VAR robtarget Openhole_5317 := [[509.38, -35.46, 190.91], [0.183051, 0.683002, 0.683002, -0.183051], [0,0,0,0], [9E9, 9E9, 9E9, 9E9, 9E9, 9E9]];
	VAR robtarget Openhole_5318 := [[536.38, -35.46, 190.83], [0.183051, 0.683002, 0.683002, -0.183051], [0,0,0,0], [9E9, 9E9, 9E9, 9E9, 9E9, 9E9]];
	VAR robtarget Openhole_5319 := [[536.38, -36.35, 191.34], [0.183051, 0.683002, 0.683002, -0.183051], [0,0,0,0], [9E9, 9E9, 9E9, 9E9, 9E9, 9E9]];
	VAR robtarget Openhole_5320 := [[509.38, -36.35, 191.42], [0.183051, 0.683002, 0.683002, -0.183051], [0,0,0,0], [9E9, 9E9, 9E9, 9E9, 9E9, 9E9]];
	VAR robtarget Openhole_5321 := [[504.38, -36.35, 190.59], [0.221198, 0.671618, 0.697002, -0.119116], [0,0,0,0], [9E9, 9E9, 9E9, 9E9, 9E9, 9E9]];
	VAR robtarget Openhole_5322 := [[504.37, -36.35, 190.59], [0.221186, 0.671622, 0.697005, -0.119099], [0,0,0,0], [9E9, 9E9, 9E9, 9E9, 9E9, 9E9]];
	VAR robtarget Openhole_5323 := [[503.88, -36.37, 190.52], [0.220113, 0.671975, 0.697256, -0.117617], [0,0,0,0], [9E9, 9E9, 9E9, 9E9, 9E9, 9E9]];
	VAR robtarget Openhole_5324 := [[492.02, -37.26, 188.91], [0.19335, 0.680159, 0.702584, -0.079844], [0,0,0,0], [9E9, 9E9, 9E9, 9E9, 9E9, 9E9]];
	VAR robtarget Openhole_5325 := [[483.16, -38.26, 187.68], [0.172338, 0.685784, 0.705428, -0.048696], [0,0,0,0], [9E9, 9E9, 9E9, 9E9, 9E9, 9E9]];
	VAR robtarget Openhole_5326 := [[480.22, -38.7, 187.26], [0.165267, 0.687522, 0.706097, -0.037783], [0,0,0,0], [9E9, 9E9, 9E9, 9E9, 9E9, 9E9]];
	VAR robtarget Openhole_5327 := [[389.31, -38.7, 170.06], [-0.126341, 0.695728, 0.665766, 0.238233], [0,0,0,0], [9E9, 9E9, 9E9, 9E9, 9E9, 9E9]];
	VAR robtarget Openhole_5328 := [[361.41, -38.7, 170.15], [-0.183051, 0.683002, 0.683002, 0.183051], [0,0,0,0], [9E9, 9E9, 9E9, 9E9, 9E9, 9E9]];
	VAR robtarget Openhole_5329 := [[362.33, -29.87, 175.24], [-0.183051, 0.683002, 0.683002, 0.183051], [0,0,0,0], [9E9, 9E9, 9E9, 9E9, 9E9, 9E9]];
	VAR robtarget Openhole_5330 := [[389.33, -29.87, 175.16], [-0.151442, 0.690699, 0.673945, 0.214006], [0,0,0,0], [9E9, 9E9, 9E9, 9E9, 9E9, 9E9]];
	VAR robtarget Openhole_5331 := [[394.33, -29.87, 175.68], [-0.137995, 0.693511, 0.677574, 0.202221], [0,0,0,0], [9E9, 9E9, 9E9, 9E9, 9E9, 9E9]];
	VAR robtarget Openhole_5332 := [[394.88, -29.88, 175.73], [-0.136468, 0.693813, 0.677964, 0.20091], [0,0,0,0], [9E9, 9E9, 9E9, 9E9, 9E9, 9E9]];
	VAR robtarget Openhole_5333 := [[399.85, -30.07, 176.16], [-0.121913, 0.696518, 0.681357, 0.189084], [0,0,0,0], [9E9, 9E9, 9E9, 9E9, 9E9, 9E9]];
	VAR robtarget Openhole_5334 := [[412.28, -31.06, 177.13], [-0.081577, 0.702385, 0.689054, 0.158759], [0,0,0,0], [9E9, 9E9, 9E9, 9E9, 9E9, 9E9]];
	VAR robtarget Openhole_5335 := [[418.24, -31.27, 177.76], [-0.061979, 0.704385, 0.69266, 0.142207], [0,0,0,0], [9E9, 9E9, 9E9, 9E9, 9E9, 9E9]];
	VAR robtarget Openhole_5336 := [[418.73, -31.27, 177.82], [-0.060379, 0.704524, 0.69296, 0.140736], [0,0,0,0], [9E9, 9E9, 9E9, 9E9, 9E9, 9E9]];
	VAR robtarget Openhole_5337 := [[423.69, -31.07, 178.45], [-0.04483, 0.705684, 0.695935, 0.125196], [0,0,0,0], [9E9, 9E9, 9E9, 9E9, 9E9, 9E9]];
	VAR robtarget Openhole_5338 := [[428.61, -30.5, 179.13], [-0.030325, 0.706456, 0.698798, 0.108078], [0,0,0,0], [9E9, 9E9, 9E9, 9E9, 9E9, 9E9]];
	VAR robtarget Openhole_5339 := [[434.95, -29.34, 179.99], [-0.012819, 0.706991, 0.702109, 0.083924], [0,0,0,0], [9E9, 9E9, 9E9, 9E9, 9E9, 9E9]];
	VAR robtarget Openhole_5340 := [[437.87, -28.76, 180.35], [-0.004854, 0.70709, 0.703391, 0.072396], [0,0,0,0], [9E9, 9E9, 9E9, 9E9, 9E9, 9E9]];
	VAR robtarget Openhole_5341 := [[438.84, -28.58, 180.46], [-0.002113, 0.707104, 0.703774, 0.068574], [0,0,0,0], [9E9, 9E9, 9E9, 9E9, 9E9, 9E9]];
	VAR robtarget Openhole_5342 := [[441.3, -28.17, 180.71], [0.004865, 0.70709, 0.704638, 0.05904], [0,0,0,0], [9E9, 9E9, 9E9, 9E9, 9E9, 9E9]];
	VAR robtarget Openhole_5343 := [[442.28, -28.03, 180.81], [0.007753, 0.707064, 0.704943, 0.055273], [0,0,0,0], [9E9, 9E9, 9E9, 9E9, 9E9, 9E9]];
	VAR robtarget Openhole_5344 := [[445.74, -27.57, 181.12], [0.017988, 0.706878, 0.705852, 0.042102], [0,0,0,0], [9E9, 9E9, 9E9, 9E9, 9E9, 9E9]];
	VAR robtarget Openhole_5345 := [[447.23, -27.43, 181.25], [0.022591, 0.706746, 0.706159, 0.036599], [0,0,0,0], [9E9, 9E9, 9E9, 9E9, 9E9, 9E9]];
	VAR robtarget Openhole_5346 := [[447.72, -27.4, 181.29], [0.024208, 0.706692, 0.706248, 0.034833], [0,0,0,0], [9E9, 9E9, 9E9, 9E9, 9E9, 9E9]];
	VAR robtarget Openhole_5347 := [[448.22, -27.39, 181.33], [0.025864, 0.706634, 0.706331, 0.033103], [0,0,0,0], [9E9, 9E9, 9E9, 9E9, 9E9, 9E9]];
	VAR robtarget Openhole_5348 := [[448.72, -27.39, 181.37], [0.027568, 0.706569, 0.706408, 0.03142], [0,0,0,0], [9E9, 9E9, 9E9, 9E9, 9E9, 9E9]];
	VAR robtarget Openhole_5349 := [[452.7, -27.62, 181.7], [0.041873, 0.705866, 0.70686, 0.018681], [0,0,0,0], [9E9, 9E9, 9E9, 9E9, 9E9, 9E9]];
	VAR robtarget Openhole_5350 := [[454.19, -27.71, 181.83], [0.047212, 0.705529, 0.70697, 0.013895], [0,0,0,0], [9E9, 9E9, 9E9, 9E9, 9E9, 9E9]];
	VAR robtarget Openhole_5351 := [[454.69, -27.73, 181.87], [0.048962, 0.70541, 0.707, 0.012271], [0,0,0,0], [9E9, 9E9, 9E9, 9E9, 9E9, 9E9]];
	VAR robtarget Openhole_5352 := [[455.68, -27.74, 181.95], [0.052367, 0.705165, 0.70705, 0.008928], [0,0,0,0], [9E9, 9E9, 9E9, 9E9, 9E9, 9E9]];
	VAR robtarget Openhole_5353 := [[456.18, -27.73, 181.99], [0.054008, 0.705041, 0.70707, 0.007198], [0,0,0,0], [9E9, 9E9, 9E9, 9E9, 9E9, 9E9]];
	VAR robtarget Openhole_5354 := [[473.12, -27.13, 183.27], [0.107256, 0.698925, 0.705213, -0.051711], [0,0,0,0], [9E9, 9E9, 9E9, 9E9, 9E9, 9E9]];
	VAR robtarget Openhole_5355 := [[498.06, -26.27, 184.82], [0.176553, 0.684711, 0.694851, -0.131083], [0,0,0,0], [9E9, 9E9, 9E9, 9E9, 9E9, 9E9]];
	VAR robtarget Openhole_5356 := [[504.36, -25.98, 185.1], [0.191702, 0.680625, 0.691162, -0.149314], [0,0,0,0], [9E9, 9E9, 9E9, 9E9, 9E9, 9E9]];
	VAR robtarget Openhole_5357 := [[509.36, -25.98, 185.43], [0.183051, 0.683002, 0.683002, -0.183051], [0,0,0,0], [9E9, 9E9, 9E9, 9E9, 9E9, 9E9]];
	VAR robtarget Openhole_5358 := [[536.36, -25.98, 185.35], [0.183051, 0.683002, 0.683002, -0.183051], [0,0,0,0], [9E9, 9E9, 9E9, 9E9, 9E9, 9E9]];
	VAR robtarget Openhole_5359 := [[536.36, -24.92, 184.74], [0.183051, 0.683002, 0.683002, -0.183051], [0,0,0,0], [9E9, 9E9, 9E9, 9E9, 9E9, 9E9]];
	VAR robtarget Openhole_5360 := [[509.36, -24.92, 184.82], [0.183051, 0.683002, 0.683002, -0.183051], [0,0,0,0], [9E9, 9E9, 9E9, 9E9, 9E9, 9E9]];
	VAR robtarget Openhole_5361 := [[504.36, -24.92, 184.54], [0.188648, 0.681478, 0.690488, -0.152403], [0,0,0,0], [9E9, 9E9, 9E9, 9E9, 9E9, 9E9]];
	VAR robtarget Openhole_5362 := [[493.09, -25.36, 184.09], [0.160531, 0.688643, 0.696924, -0.119567], [0,0,0,0], [9E9, 9E9, 9E9, 9E9, 9E9, 9E9]];
	VAR robtarget Openhole_5363 := [[469.64, -25.84, 182.75], [0.09198, 0.701099, 0.705708, -0.04446], [0,0,0,0], [9E9, 9E9, 9E9, 9E9, 9E9, 9E9]];
	VAR robtarget Openhole_5364 := [[467.64, -25.85, 182.62], [0.08559, 0.701908, 0.706096, -0.037788], [0,0,0,0], [9E9, 9E9, 9E9, 9E9, 9E9, 9E9]];
	VAR robtarget Openhole_5365 := [[467.14, -25.85, 182.59], [0.083968, 0.702104, 0.706183, -0.03613], [0,0,0,0], [9E9, 9E9, 9E9, 9E9, 9E9, 9E9]];
	VAR robtarget Openhole_5366 := [[459.66, -25.63, 182.08], [0.058601, 0.704674, 0.70701, -0.011696], [0,0,0,0], [9E9, 9E9, 9E9, 9E9, 9E9, 9E9]];
	VAR robtarget Openhole_5367 := [[455.68, -25.42, 181.81], [0.044502, 0.705705, 0.707106, 0.001108], [0,0,0,0], [9E9, 9E9, 9E9, 9E9, 9E9, 9E9]];
	VAR robtarget Openhole_5368 := [[455.18, -25.38, 181.78], [0.042678, 0.705818, 0.707102, 0.00265], [0,0,0,0], [9E9, 9E9, 9E9, 9E9, 9E9, 9E9]];
	VAR robtarget Openhole_5369 := [[454.69, -25.32, 181.74], [0.040821, 0.705928, 0.707095, 0.004156], [0,0,0,0], [9E9, 9E9, 9E9, 9E9, 9E9, 9E9]];
	VAR robtarget Openhole_5370 := [[454.1, -25.14, 181.7], [0.038206, 0.706074, 0.707085, 0.005534], [0,0,0,0], [9E9, 9E9, 9E9, 9E9, 9E9, 9E9]];
	VAR robtarget Openhole_5371 := [[451.65, -25.14, 181.56], [0.029904, 0.706474, 0.706971, 0.013856], [0,0,0,0], [9E9, 9E9, 9E9, 9E9, 9E9, 9E9]];
	VAR robtarget Openhole_5372 := [[453.08, -23.79, 181.59], [0.030159, 0.706463, 0.707093, 0.004432], [0,0,0,0], [9E9, 9E9, 9E9, 9E9, 9E9, 9E9]];
	VAR robtarget Openhole_5373 := [[455.52, -23.79, 181.7], [0.038449, 0.706061, 0.707096, -0.003884], [0,0,0,0], [9E9, 9E9, 9E9, 9E9, 9E9, 9E9]];
	VAR robtarget Openhole_5374 := [[456.08, -23.86, 181.73], [0.040591, 0.705941, 0.707085, -0.005537], [0,0,0,0], [9E9, 9E9, 9E9, 9E9, 9E9, 9E9]];
	VAR robtarget Openhole_5375 := [[457.08, -23.91, 181.78], [0.044124, 0.705729, 0.707053, -0.008753], [0,0,0,0], [9E9, 9E9, 9E9, 9E9, 9E9, 9E9]];
	VAR robtarget Openhole_5376 := [[458.58, -23.97, 181.86], [0.049362, 0.705382, 0.706976, -0.013621], [0,0,0,0], [9E9, 9E9, 9E9, 9E9, 9E9, 9E9]];
	VAR robtarget Openhole_5377 := [[465.04, -24.53, 182.25], [0.072701, 0.703359, 0.706312, -0.033524], [0,0,0,0], [9E9, 9E9, 9E9, 9E9, 9E9, 9E9]];
	VAR robtarget Openhole_5378 := [[473.03, -24.68, 182.71], [0.098941, 0.70015, 0.704603, -0.059449], [0,0,0,0], [9E9, 9E9, 9E9, 9E9, 9E9, 9E9]];
	VAR robtarget Openhole_5379 := [[473.53, -24.68, 182.74], [0.100517, 0.699926, 0.704464, -0.061077], [0,0,0,0], [9E9, 9E9, 9E9, 9E9, 9E9, 9E9]];
	VAR robtarget Openhole_5380 := [[491, -24.49, 183.61], [0.152063, 0.690563, 0.697507, -0.116122], [0,0,0,0], [9E9, 9E9, 9E9, 9E9, 9E9, 9E9]];
	VAR robtarget Openhole_5381 := [[501.99, -24.14, 184.01], [0.180425, 0.683701, 0.691377, -0.148317], [0,0,0,0], [9E9, 9E9, 9E9, 9E9, 9E9, 9E9]];
	VAR robtarget Openhole_5382 := [[504.36, -24.03, 184.07], [0.186079, 0.682184, 0.68991, -0.154997], [0,0,0,0], [9E9, 9E9, 9E9, 9E9, 9E9, 9E9]];
	VAR robtarget Openhole_5383 := [[509.36, -24.03, 184.31], [0.183051, 0.683002, 0.683002, -0.183051], [0,0,0,0], [9E9, 9E9, 9E9, 9E9, 9E9, 9E9]];
	VAR robtarget Openhole_5384 := [[536.36, -24.03, 184.23], [0.183051, 0.683002, 0.683002, -0.183051], [0,0,0,0], [9E9, 9E9, 9E9, 9E9, 9E9, 9E9]];
	VAR robtarget Openhole_5385 := [[536.35, -23.14, 183.71], [0.183051, 0.683002, 0.683002, -0.183051], [0,0,0,0], [9E9, 9E9, 9E9, 9E9, 9E9, 9E9]];
	VAR robtarget Openhole_5386 := [[509.35, -23.14, 183.8], [0.183051, 0.683002, 0.683002, -0.183051], [0,0,0,0], [9E9, 9E9, 9E9, 9E9, 9E9, 9E9]];
	VAR robtarget Openhole_5387 := [[504.35, -23.14, 183.6], [0.183484, 0.682886, 0.689318, -0.157611], [0,0,0,0], [9E9, 9E9, 9E9, 9E9, 9E9, 9E9]];
	VAR robtarget Openhole_5388 := [[494.81, -23.51, 183.38], [0.159579, 0.688865, 0.695013, -0.13022], [0,0,0,0], [9E9, 9E9, 9E9, 9E9, 9E9, 9E9]];
	VAR robtarget Openhole_5389 := [[481.32, -23.66, 182.85], [0.121281, 0.696628, 0.701446, -0.089292], [0,0,0,0], [9E9, 9E9, 9E9, 9E9, 9E9, 9E9]];
	VAR robtarget Openhole_5390 := [[480.82, -23.66, 182.82], [0.119771, 0.696889, 0.701644, -0.087728], [0,0,0,0], [9E9, 9E9, 9E9, 9E9, 9E9, 9E9]];
	VAR robtarget Openhole_5391 := [[480.32, -23.66, 182.8], [0.118257, 0.697148, 0.701838, -0.086159], [0,0,0,0], [9E9, 9E9, 9E9, 9E9, 9E9, 9E9]];
	VAR robtarget Openhole_5392 := [[479.82, -23.66, 182.78], [0.116736, 0.697404, 0.702029, -0.084589], [0,0,0,0], [9E9, 9E9, 9E9, 9E9, 9E9, 9E9]];
	VAR robtarget Openhole_5393 := [[468.84, -23.5, 182.26], [0.081646, 0.702377, 0.705366, -0.049588], [0,0,0,0], [9E9, 9E9, 9E9, 9E9, 9E9, 9E9]];
	VAR robtarget Openhole_5394 := [[463.86, -23.16, 182], [0.064212, 0.704185, 0.706282, -0.034143], [0,0,0,0], [9E9, 9E9, 9E9, 9E9, 9E9, 9E9]];
	VAR robtarget Openhole_5395 := [[459.89, -22.67, 181.79], [0.049386, 0.70538, 0.706751, -0.022432], [0,0,0,0], [9E9, 9E9, 9E9, 9E9, 9E9, 9E9]];
	VAR robtarget Openhole_5396 := [[458.89, -22.62, 181.75], [0.045863, 0.705618, 0.706845, -0.019238], [0,0,0,0], [9E9, 9E9, 9E9, 9E9, 9E9, 9E9]];
	VAR robtarget Openhole_5397 := [[457.39, -22.58, 181.7], [0.040669, 0.705936, 0.706962, -0.014321], [0,0,0,0], [9E9, 9E9, 9E9, 9E9, 9E9, 9E9]];
	VAR robtarget Openhole_5398 := [[456.89, -22.57, 181.68], [0.038969, 0.706032, 0.706994, -0.012643], [0,0,0,0], [9E9, 9E9, 9E9, 9E9, 9E9, 9E9]];
	VAR robtarget Openhole_5399 := [[456.36, -22.56, 181.66], [0.037098, 0.706133, 0.707023, -0.010873], [0,0,0,0], [9E9, 9E9, 9E9, 9E9, 9E9, 9E9]];
	VAR robtarget Openhole_5400 := [[453.91, -22.56, 181.58], [0.028813, 0.706519, 0.707102, -0.002566], [0,0,0,0], [9E9, 9E9, 9E9, 9E9, 9E9, 9E9]];
	VAR robtarget Openhole_5401 := [[454.35, -21.6, 181.55], [0.027087, 0.706588, 0.707069, -0.007307], [0,0,0,0], [9E9, 9E9, 9E9, 9E9, 9E9, 9E9]];
	VAR robtarget Openhole_5402 := [[456.8, -21.6, 181.61], [0.035372, 0.706222, 0.706935, -0.015607], [0,0,0,0], [9E9, 9E9, 9E9, 9E9, 9E9, 9E9]];
	VAR robtarget Openhole_5403 := [[457.66, -21.63, 181.63], [0.038354, 0.706066, 0.706867, -0.018425], [0,0,0,0], [9E9, 9E9, 9E9, 9E9, 9E9, 9E9]];
	VAR robtarget Openhole_5404 := [[458.15, -21.51, 181.63], [0.039592, 0.705997, 0.706811, -0.020467], [0,0,0,0], [9E9, 9E9, 9E9, 9E9, 9E9, 9E9]];
	VAR robtarget Openhole_5405 := [[458.65, -21.5, 181.64], [0.04122, 0.705904, 0.706758, -0.02221], [0,0,0,0], [9E9, 9E9, 9E9, 9E9, 9E9, 9E9]];
	VAR robtarget Openhole_5406 := [[459.15, -21.49, 181.65], [0.042898, 0.705804, 0.706703, -0.023901], [0,0,0,0], [9E9, 9E9, 9E9, 9E9, 9E9, 9E9]];
	VAR robtarget Openhole_5407 := [[459.64, -21.51, 181.67], [0.044617, 0.705698, 0.706645, -0.025546], [0,0,0,0], [9E9, 9E9, 9E9, 9E9, 9E9, 9E9]];
	VAR robtarget Openhole_5408 := [[460.14, -21.53, 181.68], [0.04638, 0.705584, 0.706586, -0.027141], [0,0,0,0], [9E9, 9E9, 9E9, 9E9, 9E9, 9E9]];
	VAR robtarget Openhole_5409 := [[461.64, -21.66, 181.73], [0.051807, 0.705206, 0.706394, -0.031736], [0,0,0,0], [9E9, 9E9, 9E9, 9E9, 9E9, 9E9]];
	VAR robtarget Openhole_5410 := [[467.1, -22.22, 181.97], [0.071741, 0.703458, 0.705467, -0.048126], [0,0,0,0], [9E9, 9E9, 9E9, 9E9, 9E9, 9E9]];
	VAR robtarget Openhole_5411 := [[475.59, -22.52, 182.3], [0.099956, 0.700006, 0.703135, -0.07484], [0,0,0,0], [9E9, 9E9, 9E9, 9E9, 9E9, 9E9]];
	VAR robtarget Openhole_5412 := [[485.58, -22.61, 182.67], [0.130652, 0.694932, 0.699149, -0.105784], [0,0,0,0], [9E9, 9E9, 9E9, 9E9, 9E9, 9E9]];
	VAR robtarget Openhole_5413 := [[486.08, -22.61, 182.69], [0.132117, 0.694655, 0.698918, -0.107301], [0,0,0,0], [9E9, 9E9, 9E9, 9E9, 9E9, 9E9]];
	VAR robtarget Openhole_5414 := [[497.58, -22.45, 183.01], [0.163867, 0.687857, 0.692854, -0.141255], [0,0,0,0], [9E9, 9E9, 9E9, 9E9, 9E9, 9E9]];
	VAR robtarget Openhole_5415 := [[504.35, -22.17, 183.08], [0.18067, 0.683636, 0.688664, -0.160441], [0,0,0,0], [9E9, 9E9, 9E9, 9E9, 9E9, 9E9]];
	VAR robtarget Openhole_5416 := [[509.35, -22.17, 183.24], [0.183051, 0.683002, 0.683002, -0.183051], [0,0,0,0], [9E9, 9E9, 9E9, 9E9, 9E9, 9E9]];
	VAR robtarget Openhole_5417 := [[536.35, -22.17, 183.15], [0.183051, 0.683002, 0.683002, -0.183051], [0,0,0,0], [9E9, 9E9, 9E9, 9E9, 9E9, 9E9]];
	VAR robtarget Openhole_5418 := [[536.35, -20.6, 182.24], [0.183051, 0.683002, 0.683002, -0.183051], [0,0,0,0], [9E9, 9E9, 9E9, 9E9, 9E9, 9E9]];
	VAR robtarget Openhole_5419 := [[509.35, -20.6, 182.33], [0.183051, 0.683002, 0.683002, -0.183051], [0,0,0,0], [9E9, 9E9, 9E9, 9E9, 9E9, 9E9]];
	VAR robtarget Openhole_5420 := [[504.35, -20.6, 182.25], [0.176089, 0.68483, 0.687578, -0.165034], [0,0,0,0], [9E9, 9E9, 9E9, 9E9, 9E9, 9E9]];
	VAR robtarget Openhole_5421 := [[495.11, -20.93, 182.26], [0.15258, 0.690449, 0.693319, -0.138954], [0,0,0,0], [9E9, 9E9, 9E9, 9E9, 9E9, 9E9]];
	VAR robtarget Openhole_5422 := [[489.11, -20.98, 182.17], [0.135831, 0.693938, 0.696595, -0.121472], [0,0,0,0], [9E9, 9E9, 9E9, 9E9, 9E9, 9E9]];
	VAR robtarget Openhole_5423 := [[488.61, -20.98, 182.16], [0.134384, 0.69422, 0.696851, -0.119997], [0,0,0,0], [9E9, 9E9, 9E9, 9E9, 9E9, 9E9]];
	VAR robtarget Openhole_5424 := [[474.12, -20.75, 181.83], [0.089526, 0.701416, 0.703021, -0.0759], [0,0,0,0], [9E9, 9E9, 9E9, 9E9, 9E9, 9E9]];
	VAR robtarget Openhole_5425 := [[464.13, -20.42, 181.62], [0.055931, 0.704891, 0.705722, -0.044224], [0,0,0,0], [9E9, 9E9, 9E9, 9E9, 9E9, 9E9]];
	VAR robtarget Openhole_5426 := [[462.63, -20.37, 181.59], [0.050745, 0.705284, 0.706007, -0.039418], [0,0,0,0], [9E9, 9E9, 9E9, 9E9, 9E9, 9E9]];
	VAR robtarget Openhole_5427 := [[461.63, -20.35, 181.58], [0.047351, 0.70552, 0.706183, -0.036123], [0,0,0,0], [9E9, 9E9, 9E9, 9E9, 9E9, 9E9]];
	VAR robtarget Openhole_5428 := [[460.13, -20.37, 181.56], [0.042403, 0.705834, 0.706427, -0.031007], [0,0,0,0], [9E9, 9E9, 9E9, 9E9, 9E9, 9E9]];
	VAR robtarget Openhole_5429 := [[459.13, -20.43, 181.55], [0.039235, 0.706017, 0.706574, -0.027456], [0,0,0,0], [9E9, 9E9, 9E9, 9E9, 9E9, 9E9]];
	VAR robtarget Openhole_5430 := [[458.63, -20.47, 181.55], [0.037695, 0.706101, 0.706642, -0.025637], [0,0,0,0], [9E9, 9E9, 9E9, 9E9, 9E9, 9E9]];
	VAR robtarget Openhole_5431 := [[457.65, -20.63, 181.55], [0.034926, 0.706244, 0.706772, -0.021748], [0,0,0,0], [9E9, 9E9, 9E9, 9E9, 9E9, 9E9]];
	VAR robtarget Openhole_5432 := [[457.1, -20.66, 181.54], [0.033189, 0.706327, 0.706829, -0.019822], [0,0,0,0], [9E9, 9E9, 9E9, 9E9, 9E9, 9E9]];
	VAR robtarget Openhole_5433 := [[454.66, -20.66, 181.5], [0.024902, 0.706668, 0.707013, -0.011531], [0,0,0,0], [9E9, 9E9, 9E9, 9E9, 9E9, 9E9]];
	VAR robtarget Openhole_5434 := [[454.85, -19.61, 181.45], [0.021982, 0.706765, 0.706932, -0.015743], [0,0,0,0], [9E9, 9E9, 9E9, 9E9, 9E9, 9E9]];
	VAR robtarget Openhole_5435 := [[457.29, -19.61, 181.47], [0.030274, 0.706458, 0.706698, -0.024026], [0,0,0,0], [9E9, 9E9, 9E9, 9E9, 9E9, 9E9]];
	VAR robtarget Openhole_5436 := [[458.04, -19.56, 181.47], [0.032606, 0.706355, 0.706602, -0.026701], [0,0,0,0], [9E9, 9E9, 9E9, 9E9, 9E9, 9E9]];
	VAR robtarget Openhole_5437 := [[460.01, -19.25, 181.44], [0.038215, 0.706073, 0.706269, -0.034403], [0,0,0,0], [9E9, 9E9, 9E9, 9E9, 9E9, 9E9]];
	VAR robtarget Openhole_5438 := [[463.44, -18.53, 181.35], [0.047252, 0.705526, 0.705456, -0.048289], [0,0,0,0], [9E9, 9E9, 9E9, 9E9, 9E9, 9E9]];
	VAR robtarget Openhole_5439 := [[464.4, -18.28, 181.31], [0.049657, 0.705361, 0.705168, -0.052331], [0,0,0,0], [9E9, 9E9, 9E9, 9E9, 9E9, 9E9]];
	VAR robtarget Openhole_5440 := [[465.37, -18.02, 181.27], [0.051958, 0.705195, 0.704853, -0.056415], [0,0,0,0], [9E9, 9E9, 9E9, 9E9, 9E9, 9E9]];
	VAR robtarget Openhole_5441 := [[467.31, -17.54, 181.16], [0.056791, 0.704823, 0.704169, -0.064395], [0,0,0,0], [9E9, 9E9, 9E9, 9E9, 9E9, 9E9]];
	VAR robtarget Openhole_5442 := [[467.8, -17.44, 181.14], [0.058071, 0.704718, 0.703989, -0.066332], [0,0,0,0], [9E9, 9E9, 9E9, 9E9, 9E9, 9E9]];
	VAR robtarget Openhole_5443 := [[468.29, -17.35, 181.12], [0.059391, 0.704608, 0.703807, -0.068237], [0,0,0,0], [9E9, 9E9, 9E9, 9E9, 9E9, 9E9]];
	VAR robtarget Openhole_5444 := [[470.26, -17.06, 181.03], [0.064904, 0.704122, 0.70305, -0.075636], [0,0,0,0], [9E9, 9E9, 9E9, 9E9, 9E9, 9E9]];
	VAR robtarget Openhole_5445 := [[471.26, -16.95, 180.98], [0.067778, 0.703851, 0.702656, -0.079209], [0,0,0,0], [9E9, 9E9, 9E9, 9E9, 9E9, 9E9]];
	VAR robtarget Openhole_5446 := [[476.25, -16.75, 180.83], [0.083173, 0.702198, 0.700589, -0.095787], [0,0,0,0], [9E9, 9E9, 9E9, 9E9, 9E9, 9E9]];
	VAR robtarget Openhole_5447 := [[478.25, -16.73, 180.78], [0.089456, 0.701425, 0.699699, -0.102084], [0,0,0,0], [9E9, 9E9, 9E9, 9E9, 9E9, 9E9]];
	VAR robtarget Openhole_5448 := [[478.75, -16.74, 180.77], [0.09103, 0.701223, 0.699471, -0.103634], [0,0,0,0], [9E9, 9E9, 9E9, 9E9, 9E9, 9E9]];
	VAR robtarget Openhole_5449 := [[491.75, -16.89, 180.55], [0.130699, 0.694923, 0.692739, -0.141821], [0,0,0,0], [9E9, 9E9, 9E9, 9E9, 9E9, 9E9]];
	VAR robtarget Openhole_5450 := [[492.25, -16.89, 180.54], [0.132135, 0.694651, 0.692447, -0.14324], [0,0,0,0], [9E9, 9E9, 9E9, 9E9, 9E9, 9E9]];
	VAR robtarget Openhole_5451 := [[500.74, -16.7, 180.27], [0.155186, 0.689868, 0.6871, -0.167015], [0,0,0,0], [9E9, 9E9, 9E9, 9E9, 9E9, 9E9]];
	VAR robtarget Openhole_5452 := [[504.34, -16.49, 180.08], [0.164104, 0.687801, 0.684601, -0.17698], [0,0,0,0], [9E9, 9E9, 9E9, 9E9, 9E9, 9E9]];
	VAR robtarget Openhole_5453 := [[509.34, -16.49, 179.96], [0.183051, 0.683002, 0.683002, -0.183051], [0,0,0,0], [9E9, 9E9, 9E9, 9E9, 9E9, 9E9]];
	VAR robtarget Openhole_5454 := [[536.34, -16.49, 179.87], [0.183051, 0.683002, 0.683002, -0.183051], [0,0,0,0], [9E9, 9E9, 9E9, 9E9, 9E9, 9E9]];
	VAR robtarget Openhole_5455 := [[536.34, -12.58, 177.62], [0.183051, 0.683002, 0.683002, -0.183051], [0,0,0,0], [9E9, 9E9, 9E9, 9E9, 9E9, 9E9]];
	VAR robtarget Openhole_5456 := [[509.34, -12.58, 177.7], [0.183051, 0.683002, 0.683002, -0.183051], [0,0,0,0], [9E9, 9E9, 9E9, 9E9, 9E9, 9E9]];
	VAR robtarget Openhole_5457 := [[504.34, -12.58, 178.01], [0.152645, 0.690434, 0.681573, -0.188305], [0,0,0,0], [9E9, 9E9, 9E9, 9E9, 9E9, 9E9]];
	VAR robtarget Openhole_5458 := [[498.82, -12.86, 178.48], [0.138448, 0.693421, 0.685524, -0.173371], [0,0,0,0], [9E9, 9E9, 9E9, 9E9, 9E9, 9E9]];
	VAR robtarget Openhole_5459 := [[495.33, -12.89, 178.71], [0.1287, 0.695296, 0.687837, -0.163953], [0,0,0,0], [9E9, 9E9, 9E9, 9E9, 9E9, 9E9]];
	VAR robtarget Openhole_5460 := [[494.83, -12.89, 178.73], [0.127263, 0.69556, 0.688156, -0.162606], [0,0,0,0], [9E9, 9E9, 9E9, 9E9, 9E9, 9E9]];
	VAR robtarget Openhole_5461 := [[482.35, -12.7, 179.41], [0.089272, 0.701449, 0.69551, -0.127536], [0,0,0,0], [9E9, 9E9, 9E9, 9E9, 9E9, 9E9]];
	VAR robtarget Openhole_5462 := [[481.85, -12.7, 179.44], [0.08772, 0.701645, 0.695784, -0.126035], [0,0,0,0], [9E9, 9E9, 9E9, 9E9, 9E9, 9E9]];
	VAR robtarget Openhole_5463 := [[476.37, -12.88, 179.82], [0.07088, 0.703545, 0.698695, -0.108745], [0,0,0,0], [9E9, 9E9, 9E9, 9E9, 9E9, 9E9]];
	VAR robtarget Openhole_5464 := [[472.41, -13.34, 180.16], [0.059569, 0.704593, 0.700723, -0.094801], [0,0,0,0], [9E9, 9E9, 9E9, 9E9, 9E9, 9E9]];
	VAR robtarget Openhole_5465 := [[471.92, -13.42, 180.2], [0.058232, 0.704705, 0.700968, -0.09297], [0,0,0,0], [9E9, 9E9, 9E9, 9E9, 9E9, 9E9]];
	VAR robtarget Openhole_5466 := [[470.94, -13.62, 180.3], [0.055684, 0.704911, 0.701458, -0.089204], [0,0,0,0], [9E9, 9E9, 9E9, 9E9, 9E9, 9E9]];
	VAR robtarget Openhole_5467 := [[470.46, -13.73, 180.34], [0.054453, 0.705007, 0.701699, -0.087285], [0,0,0,0], [9E9, 9E9, 9E9, 9E9, 9E9, 9E9]];
	VAR robtarget Openhole_5468 := [[469.49, -13.97, 180.44], [0.052075, 0.705187, 0.702174, -0.083378], [0,0,0,0], [9E9, 9E9, 9E9, 9E9, 9E9, 9E9]];
	VAR robtarget Openhole_5469 := [[468.53, -14.24, 180.54], [0.04981, 0.70535, 0.702637, -0.079383], [0,0,0,0], [9E9, 9E9, 9E9, 9E9, 9E9, 9E9]];
	VAR robtarget Openhole_5470 := [[467.59, -14.54, 180.63], [0.04769, 0.705497, 0.703087, -0.075291], [0,0,0,0], [9E9, 9E9, 9E9, 9E9, 9E9, 9E9]];
	VAR robtarget Openhole_5471 := [[467.12, -14.71, 180.68], [0.046691, 0.705564, 0.703307, -0.073207], [0,0,0,0], [9E9, 9E9, 9E9, 9E9, 9E9, 9E9]];
	VAR robtarget Openhole_5472 := [[466.65, -14.89, 180.73], [0.04574, 0.705626, 0.703523, -0.071096], [0,0,0,0], [9E9, 9E9, 9E9, 9E9, 9E9, 9E9]];
	VAR robtarget Openhole_5473 := [[466.19, -15.08, 180.78], [0.044843, 0.705683, 0.703736, -0.068958], [0,0,0,0], [9E9, 9E9, 9E9, 9E9, 9E9, 9E9]];
	VAR robtarget Openhole_5474 := [[465.74, -15.28, 180.83], [0.043986, 0.705737, 0.703945, -0.066798], [0,0,0,0], [9E9, 9E9, 9E9, 9E9, 9E9, 9E9]];
	VAR robtarget Openhole_5475 := [[464.83, -15.7, 180.93], [0.042389, 0.705835, 0.704346, -0.062422], [0,0,0,0], [9E9, 9E9, 9E9, 9E9, 9E9, 9E9]];
	VAR robtarget Openhole_5476 := [[463.94, -16.14, 181.02], [0.040919, 0.705922, 0.704726, -0.057982], [0,0,0,0], [9E9, 9E9, 9E9, 9E9, 9E9, 9E9]];
	VAR robtarget Openhole_5477 := [[462.19, -17.09, 181.18], [0.03822, 0.706073, 0.705409, -0.048978], [0,0,0,0], [9E9, 9E9, 9E9, 9E9, 9E9, 9E9]];
	VAR robtarget Openhole_5478 := [[461.3, -17.54, 181.25], [0.036782, 0.706149, 0.705706, -0.04448], [0,0,0,0], [9E9, 9E9, 9E9, 9E9, 9E9, 9E9]];
	VAR robtarget Openhole_5479 := [[460.84, -17.74, 181.28], [0.035885, 0.706196, 0.705841, -0.042289], [0,0,0,0], [9E9, 9E9, 9E9, 9E9, 9E9, 9E9]];
	VAR robtarget Openhole_5480 := [[460.38, -17.92, 181.3], [0.034933, 0.706243, 0.705968, -0.040118], [0,0,0,0], [9E9, 9E9, 9E9, 9E9, 9E9, 9E9]];
	VAR robtarget Openhole_5481 := [[459.42, -18.22, 181.34], [0.032729, 0.706349, 0.706194, -0.035909], [0,0,0,0], [9E9, 9E9, 9E9, 9E9, 9E9, 9E9]];
	VAR robtarget Openhole_5482 := [[458.45, -18.46, 181.37], [0.030283, 0.706458, 0.70639, -0.031823], [0,0,0,0], [9E9, 9E9, 9E9, 9E9, 9E9, 9E9]];
	VAR robtarget Openhole_5483 := [[457.96, -18.57, 181.38], [0.029004, 0.706512, 0.706478, -0.02981], [0,0,0,0], [9E9, 9E9, 9E9, 9E9, 9E9, 9E9]];
	VAR robtarget Openhole_5484 := [[457.35, -18.58, 181.39], [0.026933, 0.706594, 0.706564, -0.027702], [0,0,0,0], [9E9, 9E9, 9E9, 9E9, 9E9, 9E9]];
	VAR robtarget Openhole_5485 := [[454.9, -18.58, 181.4], [0.018635, 0.706861, 0.70684, -0.019426], [0,0,0,0], [9E9, 9E9, 9E9, 9E9, 9E9, 9E9]];
	VAR robtarget Openhole_5486 := [[454.82, -17.6, 181.35], [0.015053, 0.706947, 0.706749, -0.022484], [0,0,0,0], [9E9, 9E9, 9E9, 9E9, 9E9, 9E9]];
	VAR robtarget Openhole_5487 := [[457.27, -17.6, 181.31], [0.023358, 0.706721, 0.706438, -0.030755], [0,0,0,0], [9E9, 9E9, 9E9, 9E9, 9E9, 9E9]];
	VAR robtarget Openhole_5488 := [[457.88, -17.43, 181.29], [0.024867, 0.706669, 0.706318, -0.033386], [0,0,0,0], [9E9, 9E9, 9E9, 9E9, 9E9, 9E9]];
	VAR robtarget Openhole_5489 := [[458.35, -17.26, 181.27], [0.025881, 0.706633, 0.706213, -0.035542], [0,0,0,0], [9E9, 9E9, 9E9, 9E9, 9E9, 9E9]];
	VAR robtarget Openhole_5490 := [[458.82, -17.08, 181.24], [0.026837, 0.706597, 0.7061, -0.037721], [0,0,0,0], [9E9, 9E9, 9E9, 9E9, 9E9, 9E9]];
	VAR robtarget Openhole_5491 := [[459.27, -16.88, 181.22], [0.027686, 0.706565, 0.705978, -0.039941], [0,0,0,0], [9E9, 9E9, 9E9, 9E9, 9E9, 9E9]];
	VAR robtarget Openhole_5492 := [[459.72, -16.65, 181.18], [0.028442, 0.706535, 0.705847, -0.04219], [0,0,0,0], [9E9, 9E9, 9E9, 9E9, 9E9, 9E9]];
	VAR robtarget Openhole_5493 := [[460.15, -16.4, 181.15], [0.029036, 0.70651, 0.705706, -0.044484], [0,0,0,0], [9E9, 9E9, 9E9, 9E9, 9E9, 9E9]];
	VAR robtarget Openhole_5494 := [[461.82, -15.31, 180.98], [0.030996, 0.706427, 0.705063, -0.053717], [0,0,0,0], [9E9, 9E9, 9E9, 9E9, 9E9, 9E9]];
	VAR robtarget Openhole_5495 := [[463.11, -14.56, 180.83], [0.032806, 0.706345, 0.704512, -0.060521], [0,0,0,0], [9E9, 9E9, 9E9, 9E9, 9E9, 9E9]];
	VAR robtarget Openhole_5496 := [[464.88, -13.66, 180.62], [0.035704, 0.706205, 0.703694, -0.069391], [0,0,0,0], [9E9, 9E9, 9E9, 9E9, 9E9, 9E9]];
	VAR robtarget Openhole_5497 := [[465.33, -13.45, 180.56], [0.036526, 0.706163, 0.703476, -0.071563], [0,0,0,0], [9E9, 9E9, 9E9, 9E9, 9E9, 9E9]];
	VAR robtarget Openhole_5498 := [[465.79, -13.26, 180.51], [0.037406, 0.706117, 0.703255, -0.073709], [0,0,0,0], [9E9, 9E9, 9E9, 9E9, 9E9, 9E9]];
	VAR robtarget Openhole_5499 := [[466.25, -13.07, 180.45], [0.038332, 0.706067, 0.703029, -0.07583], [0,0,0,0], [9E9, 9E9, 9E9, 9E9, 9E9, 9E9]];
	VAR robtarget Openhole_5500 := [[467.66, -12.58, 180.28], [0.041359, 0.705896, 0.70233, -0.082053], [0,0,0,0], [9E9, 9E9, 9E9, 9E9, 9E9, 9E9]];
	VAR robtarget Openhole_5501 := [[468.61, -12.29, 180.17], [0.04355, 0.705764, 0.701847, -0.08609], [0,0,0,0], [9E9, 9E9, 9E9, 9E9, 9E9, 9E9]];
	VAR robtarget Openhole_5502 := [[469.57, -12.03, 180.06], [0.045867, 0.705618, 0.701351, -0.090035], [0,0,0,0], [9E9, 9E9, 9E9, 9E9, 9E9, 9E9]];
	VAR robtarget Openhole_5503 := [[470.53, -11.8, 179.95], [0.048309, 0.705455, 0.700846, -0.093884], [0,0,0,0], [9E9, 9E9, 9E9, 9E9, 9E9, 9E9]];
	VAR robtarget Openhole_5504 := [[471.02, -11.7, 179.89], [0.049576, 0.705367, 0.700591, -0.095771], [0,0,0,0], [9E9, 9E9, 9E9, 9E9, 9E9, 9E9]];
	VAR robtarget Openhole_5505 := [[474.95, -11.1, 179.47], [0.060501, 0.704514, 0.698483, -0.110096], [0,0,0,0], [9E9, 9E9, 9E9, 9E9, 9E9, 9E9]];
	VAR robtarget Openhole_5506 := [[478.92, -10.84, 179.09], [0.072468, 0.703384, 0.6963, -0.123149], [0,0,0,0], [9E9, 9E9, 9E9, 9E9, 9E9, 9E9]];
	VAR robtarget Openhole_5507 := [[482.41, -10.79, 178.8], [0.08335, 0.702177, 0.694337, -0.133777], [0,0,0,0], [9E9, 9E9, 9E9, 9E9, 9E9, 9E9]];
	VAR robtarget Openhole_5508 := [[482.91, -10.8, 178.76], [0.084919, 0.701989, 0.694052, -0.135245], [0,0,0,0], [9E9, 9E9, 9E9, 9E9, 9E9, 9E9]];
	VAR robtarget Openhole_5509 := [[497.37, -11.14, 177.78], [0.129205, 0.695202, 0.685195, -0.174664], [0,0,0,0], [9E9, 9E9, 9E9, 9E9, 9E9, 9E9]];
	VAR robtarget Openhole_5510 := [[497.87, -11.14, 177.74], [0.130614, 0.694939, 0.684859, -0.175978], [0,0,0,0], [9E9, 9E9, 9E9, 9E9, 9E9, 9E9]];
	VAR robtarget Openhole_5511 := [[502.85, -10.99, 177.28], [0.143939, 0.692302, 0.681322, -0.189209], [0,0,0,0], [9E9, 9E9, 9E9, 9E9, 9E9, 9E9]];
	VAR robtarget Openhole_5512 := [[504.39, -10.89, 177.11], [0.147831, 0.691481, 0.680161, -0.193342], [0,0,0,0], [9E9, 9E9, 9E9, 9E9, 9E9, 9E9]];
	VAR robtarget Openhole_5513 := [[509.33, -10.89, 176.72], [0.183051, 0.683002, 0.683002, -0.183051], [0,0,0,0], [9E9, 9E9, 9E9, 9E9, 9E9, 9E9]];
	VAR robtarget Openhole_5514 := [[536.33, -10.89, 176.64], [0.183051, 0.683002, 0.683002, -0.183051], [0,0,0,0], [9E9, 9E9, 9E9, 9E9, 9E9, 9E9]];
	VAR robtarget Openhole_5515 := [[536.33, -10, 176.13], [0.183051, 0.683002, 0.683002, -0.183051], [0,0,0,0], [9E9, 9E9, 9E9, 9E9, 9E9, 9E9]];
	VAR robtarget Openhole_5516 := [[509.33, -10, 176.21], [0.183051, 0.683002, 0.683002, -0.183051], [0,0,0,0], [9E9, 9E9, 9E9, 9E9, 9E9, 9E9]];
	VAR robtarget Openhole_5517 := [[504.33, -10, 176.65], [0.14508, 0.692063, 0.679477, -0.19573], [0,0,0,0], [9E9, 9E9, 9E9, 9E9, 9E9, 9E9]];
	VAR robtarget Openhole_5518 := [[503.56, -10.02, 176.72], [0.143018, 0.692492, 0.680037, -0.193777], [0,0,0,0], [9E9, 9E9, 9E9, 9E9, 9E9, 9E9]];
	VAR robtarget Openhole_5519 := [[499.58, -10.13, 177.12], [0.132364, 0.694608, 0.682904, -0.183418], [0,0,0,0], [9E9, 9E9, 9E9, 9E9, 9E9, 9E9]];
	VAR robtarget Openhole_5520 := [[499.08, -10.12, 177.16], [0.130958, 0.694874, 0.683246, -0.18214], [0,0,0,0], [9E9, 9E9, 9E9, 9E9, 9E9, 9E9]];
	VAR robtarget Openhole_5521 := [[490.61, -9.87, 177.78], [0.105574, 0.699181, 0.688723, -0.160189], [0,0,0,0], [9E9, 9E9, 9E9, 9E9, 9E9, 9E9]];
